BEGIN
   MachineConfig[0].Machine."Family" := 2;
   MachineConfig[0].Machine.TypeNo := 20;
   MachineConfig[0].Machine.Range := 2;
   MachineConfig[0].Machine.SepType := 1;
   MachineConfig[0].Machine.Frame := 4;
   MachineConfig[0].Machine.DchSystem := 1;
   MachineConfig[0].Machine.Spare_1 := 3;
   MachineConfig[0].Machine.FeedPump := 1;
   MachineConfig[0].Machine.eWON := 1;
   MachineConfig[0]."Unit Sep"."EM - 100"."L-GREEN".CW.ENABLE := TRUE;
   MachineConfig[0]."Unit Sep"."EM - 100"."L-YELLOW".Tag := 'L-BLUE';
   MachineConfig[0]."Unit Sep"."EM - 100".EMS.Address := 180;
   MachineConfig[0]."Unit Sep"."EM - 100".UPS.CW.ENABLE := False;
   MachineConfig[0]."Unit Sep"."EM - 100".EWON.CW.ENABLE := True;
   MachineConfig[0]."Unit Sep"."EM - 100".EWON.CW.EXIST := True;
   MachineConfig[0]."Unit Sep"."EM - 100"."LT BUF".CW.ENABLE := False;
   MachineConfig[0]."Unit Sep"."EM - 400"."AV409-1".CW.ENABLE := False;
   MachineConfig[0]."Unit Sep"."EM - 400"."AV409-1".ACT_OUT_ADD := 8;
   MachineConfig[0]."Unit Sep"."EM - 400"."FCV409-1".CW.ENABLE := False;
   MachineConfig[0]."Unit Sep"."EM - 400"."FIS409-1".CW.ENABLE := false;
   MachineConfig[0]."Unit Sep"."EM - 400"."FIT409-1".CW.ENABLE := False;
   MachineConfig[0]."Unit Sep"."EM - 701".M701."TYPE" := 2;
   MachineConfig[0]."Unit Sep"."EM - 701".M701.FB_RUN_ADD := 8;
   MachineConfig[0]."Unit Sep"."EM - 701".M701.FB_RDY_ADD := 8;
   MachineConfig[0]."Unit Sep"."EM - 701".M701.OUT_ACT_ADD := 512;
   MachineConfig[0]."Unit Sep"."EM - 701".M701.OUT_RST_ADD := 8;
   MachineConfig[0]."Unit Sep"."EM - 730".TS730.CW.ENABLE := True;
   MachineConfig[0]."Unit Sep"."EM - 730".TS730.Address := 184;
   MachineConfig[0]."Unit Sep"."EM - 740"."P+F PS".Address := 180;
   MachineConfig[0]."Unit Sep"."EM - 740"."P+F OS".Address := 182;
   MachineConfig[0]."Unit Sep"."EM - 740"."P+F ERROR".Address := 183;
   MachineConfig[0]."Unit Sep"."EM - 750".YT75X.CW.ENABLE := False;
   MachineConfig[0]."Unit Process"."EM - 201"."AV201-1".CW.ENABLE := True;
   MachineConfig[0]."Unit Process"."EM - 201"."AV201-1".CW.FB_CLS_EN := False;
   MachineConfig[0]."Unit Process"."EM - 201"."AV201-1".CW.FB_OPN_EN := False;
   MachineConfig[0]."Unit Process"."EM - 201"."AV201-1".CW.VLV_W_FB := False;
   MachineConfig[0]."Unit Process"."EM - 201"."AV201-1".FB_OPN_ADD := 8;
   MachineConfig[0]."Unit Process"."EM - 201"."AV201-1".FB_CLS_ADD := 8;
   MachineConfig[0]."Unit Process"."EM - 201"."AV201-1".ACT_OUT_ADD := 160;
   MachineConfig[0]."Unit Process"."EM - 201"."FCV201-1".CW.ENABLE := false;
   MachineConfig[0]."Unit Process"."EM - 201"."FIT201-1"."Type" := 0;
   MachineConfig[0]."Unit Process"."EM - 201"."FIT201-1".Address := 88;
   MachineConfig[0]."Unit Process"."EM - 201"."FIT201-1".Max := 10000.0;
   MachineConfig[0]."Unit Process"."EM - 201"."LA201-1".CW.ENABLE := False;
   MachineConfig[0]."Unit Process"."EM - 201"."PIT201-1".CW.ENABLE := False;
   MachineConfig[0]."Unit Process"."EM - 22X"."AV220-1".CW.ENABLE := True;
   MachineConfig[0]."Unit Process"."EM - 22X"."AV220-1".CW.FB_CLS_EN := false;
   MachineConfig[0]."Unit Process"."EM - 22X"."AV220-1".CW.FB_OPN_EN := false;
   MachineConfig[0]."Unit Process"."EM - 22X"."AV220-1".CW.EXIST := False;
   MachineConfig[0]."Unit Process"."EM - 22X"."AV220-1".CW.VLV_W_FB := false;
   MachineConfig[0]."Unit Process"."EM - 22X"."AV220-1".FB_OPN_ADD := 8;
   MachineConfig[0]."Unit Process"."EM - 22X"."AV220-1".FB_CLS_ADD := 8;
   MachineConfig[0]."Unit Process"."EM - 22X"."AV220-1".ACT_OUT_ADD := 162;
   MachineConfig[0]."Unit Process"."EM - 22X"."AV460-1".CW.ENABLE := True;
   MachineConfig[0]."Unit Process"."EM - 22X"."AV460-1".CW.FB_CLS_EN := false;
   MachineConfig[0]."Unit Process"."EM - 22X"."AV460-1".CW.FB_OPN_EN := false;
   MachineConfig[0]."Unit Process"."EM - 22X"."AV460-1".CW.EXIST := False;
   MachineConfig[0]."Unit Process"."EM - 22X"."AV460-1".CW.VLV_W_FB := false;
   MachineConfig[0]."Unit Process"."EM - 22X"."AV460-1".FB_OPN_ADD := 8;
   MachineConfig[0]."Unit Process"."EM - 22X"."AV460-1".FB_CLS_ADD := 8;
   MachineConfig[0]."Unit Process"."EM - 22X"."AV460-1".ACT_OUT_ADD := 171;
   MachineConfig[0]."Unit Process"."EM - 22X"."FIT22X-1".CW.ENABLE := False;
   MachineConfig[0]."Unit Process"."EM - 22X"."PIT22X-1".CW.ENABLE := False;
   MachineConfig[0]."Unit Process"."EM - 22X"."PIT22X-1".CW.EXIST := False;
   MachineConfig[0]."Unit Process"."EM - 22X"."QT220-1".Tag := 'QT220-1';
   MachineConfig[0]."Unit Process"."EM - 22X"."QT220-1".CW.ENABLE := True;
   MachineConfig[0]."Unit Process"."EM - 22X"."QT220-1".CW.EXIST := False;
   MachineConfig[0]."Unit Process"."EM - 22X"."QT220-1".Address := 70;
   MachineConfig[0]."Unit Process"."EM - 22X"."PCV22X-1".CW.ENABLE := False;
   MachineConfig[0]."Unit Process"."EM - 22Y"."AV221-1".CW.ENABLE := false;
   MachineConfig[0]."Unit Process"."EM - 22Y"."AV461-1".CW.ENABLE := false;
   MachineConfig[0]."Unit Process"."EM - 22Y"."FIT22Y-1".CW.ENABLE := false;
   MachineConfig[0]."Unit Process"."EM - 22Y"."LA221-1".CW.ENABLE := false;
   MachineConfig[0]."Unit Process"."EM - 22Y"."PCV22Y-1".CW.ENABLE := false;
   MachineConfig[0]."Unit Process"."EM - 22Y"."PIT22Y-1".CW.ENABLE := false;
   MachineConfig[0]."Unit Process"."EM - 340"."AV340-1".CW.ENABLE := True;
   MachineConfig[0]."Unit Process"."EM - 340"."AV340-1".CW.FB_CLS_EN := False;
   MachineConfig[0]."Unit Process"."EM - 340"."AV340-1".CW.FB_OPN_EN := False;
   MachineConfig[0]."Unit Process"."EM - 340"."AV340-1".CW.EXIST := False;
   MachineConfig[0]."Unit Process"."EM - 340"."AV340-1".CW.VLV_W_FB := False;
   MachineConfig[0]."Unit Process"."EM - 340"."AV340-1".FB_OPN_ADD := 8;
   MachineConfig[0]."Unit Process"."EM - 340"."AV340-1".FB_CLS_ADD := 8;
   MachineConfig[0]."Unit Process"."EM - 340"."AV340-1".ACT_OUT_ADD := 165;
   MachineConfig[0]."Unit Process"."EM - 340"."PIS340-1".Tag := 'PS301-1';
   MachineConfig[0]."Unit Process"."EM - 340"."PIS340-1".CW.ENABLE := True;
   MachineConfig[0]."Unit Process"."EM - 340"."V340-1".CW.ENABLE := True;
   MachineConfig[0]."Unit Process"."EM - 340"."V340-1".Address := 170;
   MachineConfig[0]."Unit Dch"."EM - 222"."LS222-1".CW.ENABLE := False;
   MachineConfig[0]."Unit Dch"."EM - 222"."P222-1".CW.EXIST := False;
   MachineConfig[0]."Unit Dch"."EM - 222"."P222-1".FB_RUN_ADD := 194;
   MachineConfig[0]."Unit Dch"."EM - 222"."P222-1".FB_RDY_ADD := 195;
   MachineConfig[0]."Unit Dch"."EM - 222"."P222-1".OUT_ACT_ADD := 182;
   MachineConfig[0]."Unit Dch"."EM - 222"."TS222-1".CW.ENABLE := false;
   MachineConfig[0]."Unit Dch"."EM - 300"."AV301-1".CW.ENABLE := True;
   MachineConfig[0]."Unit Dch"."EM - 300"."AV301-1".CW.FB_CLS_EN := false;
   MachineConfig[0]."Unit Dch"."EM - 300"."AV301-1".CW.FB_OPN_EN := false;
   MachineConfig[0]."Unit Dch"."EM - 300"."AV301-1".CW.VLV_W_FB := false;
   MachineConfig[0]."Unit Dch"."EM - 300"."AV301-1".FB_OPN_ADD := 8;
   MachineConfig[0]."Unit Dch"."EM - 300"."AV301-1".FB_CLS_ADD := 8;
   MachineConfig[0]."Unit Dch"."EM - 300"."AV301-1".ACT_OUT_ADD := 163;
   MachineConfig[0]."Unit Dch"."EM - 300"."AV304-1".TAG := 'AV301-1';
   MachineConfig[0]."Unit Dch"."EM - 300"."AV304-1".ACT_OUT_ADD := 163;
   MachineConfig[0]."Unit Dch"."EM - 300"."AV320-1".CW.ENABLE := True;
   MachineConfig[0]."Unit Dch"."EM - 300"."AV320-1".CW.FB_CLS_EN := false;
   MachineConfig[0]."Unit Dch"."EM - 300"."AV320-1".CW.FB_OPN_EN := false;
   MachineConfig[0]."Unit Dch"."EM - 300"."AV320-1".CW.EXIST := false;
   MachineConfig[0]."Unit Dch"."EM - 300"."AV320-1".CW.VLV_W_FB := false;
   MachineConfig[0]."Unit Dch"."EM - 300"."AV320-1".FB_OPN_ADD := 8;
   MachineConfig[0]."Unit Dch"."EM - 300"."AV320-1".FB_CLS_ADD := 8;
   MachineConfig[0]."Unit Dch"."EM - 300"."AV320-1".ACT_OUT_ADD := 164;
   MachineConfig[0]."Unit Dch"."EM - 300"."PS301-1".CW.ENABLE := True;
   MachineConfig[0]."Unit Dch"."EM - 375"."AV37X-1".TAG := 'AV376-1';
   MachineConfig[0]."Unit Dch"."EM - 375"."AV37X-1".CW.ENABLE := true;
   MachineConfig[0]."Unit Dch"."EM - 375"."AV37X-1".ACT_OUT_ADD := 166;
   MachineConfig[0]."Unit Dch"."EM - 375".LS793.CW.ENABLE := true;
   MachineConfig[0]."Unit Dch"."EM - 375"."PIS375-1".CW.ENABLE := false;
   MachineConfig[0]."Unit Dch"."EM - 506".IP506a.CW.ENABLE := False;
   MachineConfig[0]."Unit Dch"."EM - 506".AVDCH.TAG := 'AV372-1';
   MachineConfig[0]."Unit Dch"."EM - 506".AVDCH.CW.ENABLE := true;
   MachineConfig[0]."Unit Dch"."EM - 506".AVDCH.ACT_OUT_ADD := 167;
   MachineConfig[0].Options."EM - P201"."P201-1".FB_RUN_ADD := 196;
   MachineConfig[0].Options."EM - P201"."P201-1".FB_RDY_ADD := 197;
   MachineConfig[0].Options."EM - P201"."P201-1".OUT_ACT_ADD := 183;
   MachineConfig[0].Options."EM - P201"."P201-1".OUT_RST_ADD := 184;
   MachineConfig[0].Options."EM - P201"."P201-1_SPEED_REF".Address := 70;
   MachineConfig[1].Machine."Family" := 2;
   MachineConfig[1].Machine.TypeNo := 21;
   MachineConfig[1].Machine.Range := 2;
   MachineConfig[1].Machine.SepType := 2;
   MachineConfig[1].Machine.Frame := 4;
   MachineConfig[1].Machine.DchSystem := 1;
   MachineConfig[1].Machine.Spare_1 := 3;
   MachineConfig[1].Machine.FeedPump := 1;
   MachineConfig[1].Machine.eWON := 1;
   MachineConfig[1]."Unit Sep"."EM - 100"."L-GREEN".CW.ENABLE := True;
   MachineConfig[1]."Unit Sep"."EM - 100"."L-YELLOW".Tag := 'L-BLUE';
   MachineConfig[1]."Unit Sep"."EM - 100".EMS.Address := 180;
   MachineConfig[1]."Unit Sep"."EM - 100".UPS.CW.ENABLE := False;
   MachineConfig[1]."Unit Sep"."EM - 100".EWON.CW.ENABLE := True;
   MachineConfig[1]."Unit Sep"."EM - 100".EWON.CW.EXIST := True;
   MachineConfig[1]."Unit Sep"."EM - 100"."LT BUF".CW.ENABLE := False;
   MachineConfig[1]."Unit Sep"."EM - 400"."AV409-1".CW.ENABLE := False;
   MachineConfig[1]."Unit Sep"."EM - 400"."FCV409-1".CW.ENABLE := False;
   MachineConfig[1]."Unit Sep"."EM - 400"."FIS409-1".CW.ENABLE := false;
   MachineConfig[1]."Unit Sep"."EM - 400"."FIT409-1".CW.ENABLE := False;
   MachineConfig[1]."Unit Sep"."EM - 701".M701."TYPE" := 2;
   MachineConfig[1]."Unit Sep"."EM - 701".M701.FB_RUN_ADD := 8;
   MachineConfig[1]."Unit Sep"."EM - 701".M701.FB_RDY_ADD := 8;
   MachineConfig[1]."Unit Sep"."EM - 701".M701.OUT_ACT_ADD := 512;
   MachineConfig[1]."Unit Sep"."EM - 701".M701.OUT_RST_ADD := 8;
   MachineConfig[1]."Unit Sep"."EM - 730".TS730.CW.ENABLE := True;
   MachineConfig[1]."Unit Sep"."EM - 730".TS730.Address := 184;
   MachineConfig[1]."Unit Sep"."EM - 740"."P+F PS".Address := 180;
   MachineConfig[1]."Unit Sep"."EM - 740"."P+F OS".Address := 182;
   MachineConfig[1]."Unit Sep"."EM - 740"."P+F ERROR".Address := 183;
   MachineConfig[1]."Unit Sep"."EM - 750".YT75X.CW.ENABLE := False;
   MachineConfig[1]."Unit Process"."EM - 201"."AV201-1".CW.ENABLE := True;
   MachineConfig[1]."Unit Process"."EM - 201"."AV201-1".CW.VLV_W_FB := false;
   MachineConfig[1]."Unit Process"."EM - 201"."AV201-1".FB_OPN_ADD := 8;
   MachineConfig[1]."Unit Process"."EM - 201"."AV201-1".FB_CLS_ADD := 8;
   MachineConfig[1]."Unit Process"."EM - 201"."AV201-1".ACT_OUT_ADD := 160;
   MachineConfig[1]."Unit Process"."EM - 201"."FCV201-1".CW.ENABLE := false;
   MachineConfig[1]."Unit Process"."EM - 201"."FIT201-1"."Type" := 0;
   MachineConfig[1]."Unit Process"."EM - 201"."FIT201-1".Address := 88;
   MachineConfig[1]."Unit Process"."EM - 201"."FIT201-1".Max := 10000.0;
   MachineConfig[1]."Unit Process"."EM - 201"."LA201-1".CW.ENABLE := False;
   MachineConfig[1]."Unit Process"."EM - 201"."PIT201-1".CW.ENABLE := False;
   MachineConfig[1]."Unit Process"."EM - 22X"."FIT22X-1".CW.ENABLE := False;
   MachineConfig[1]."Unit Process"."EM - 22X"."PIT22X-1".CW.ENABLE := False;
   MachineConfig[1]."Unit Process"."EM - 22X"."PCV22X-1".CW.ENABLE := False;
   MachineConfig[1]."Unit Process"."EM - 22Y"."AV221-1".CW.ENABLE := True;
   MachineConfig[1]."Unit Process"."EM - 22Y"."AV221-1".CW.FB_CLS_EN := false;
   MachineConfig[1]."Unit Process"."EM - 22Y"."AV221-1".CW.FB_OPN_EN := false;
   MachineConfig[1]."Unit Process"."EM - 22Y"."AV221-1".CW.EXIST := false;
   MachineConfig[1]."Unit Process"."EM - 22Y"."AV221-1".CW.VLV_W_FB := false;
   MachineConfig[1]."Unit Process"."EM - 22Y"."AV221-1".FB_OPN_ADD := 8;
   MachineConfig[1]."Unit Process"."EM - 22Y"."AV221-1".FB_CLS_ADD := 8;
   MachineConfig[1]."Unit Process"."EM - 22Y"."AV221-1".ACT_OUT_ADD := 175;
   MachineConfig[1]."Unit Process"."EM - 22Y"."AV461-1".CW.ENABLE := True;
   MachineConfig[1]."Unit Process"."EM - 22Y"."AV461-1".CW.FB_CLS_EN := false;
   MachineConfig[1]."Unit Process"."EM - 22Y"."AV461-1".CW.FB_OPN_EN := false;
   MachineConfig[1]."Unit Process"."EM - 22Y"."AV461-1".CW.EXIST := false;
   MachineConfig[1]."Unit Process"."EM - 22Y"."AV461-1".CW.VLV_W_FB := false;
   MachineConfig[1]."Unit Process"."EM - 22Y"."AV461-1".FB_OPN_ADD := 8;
   MachineConfig[1]."Unit Process"."EM - 22Y"."AV461-1".FB_CLS_ADD := 8;
   MachineConfig[1]."Unit Process"."EM - 22Y"."AV461-1".ACT_OUT_ADD := 176;
   MachineConfig[1]."Unit Process"."EM - 340"."AV340-1".CW.FB_CLS_EN := False;
   MachineConfig[1]."Unit Process"."EM - 340"."AV340-1".CW.FB_OPN_EN := False;
   MachineConfig[1]."Unit Process"."EM - 340"."AV340-1".CW.EXIST := False;
   MachineConfig[1]."Unit Process"."EM - 340"."AV340-1".CW.VLV_W_FB := False;
   MachineConfig[1]."Unit Process"."EM - 340"."AV340-1".FB_OPN_ADD := 8;
   MachineConfig[1]."Unit Process"."EM - 340"."AV340-1".FB_CLS_ADD := 8;
   MachineConfig[1]."Unit Process"."EM - 340"."AV340-1".ACT_OUT_ADD := 165;
   MachineConfig[1]."Unit Process"."EM - 340"."PIS340-1".Tag := 'PS301-1';
   MachineConfig[1]."Unit Process"."EM - 340"."PIS340-1".CW.ENABLE := True;
   MachineConfig[1]."Unit Dch"."EM - 222"."LS222-1".CW.ENABLE := False;
   MachineConfig[1]."Unit Dch"."EM - 222"."P222-1".CW.EXIST := False;
   MachineConfig[1]."Unit Dch"."EM - 222"."P222-1".FB_RUN_ADD := 194;
   MachineConfig[1]."Unit Dch"."EM - 222"."P222-1".FB_RDY_ADD := 195;
   MachineConfig[1]."Unit Dch"."EM - 222"."P222-1".OUT_ACT_ADD := 182;
   MachineConfig[1]."Unit Dch"."EM - 222"."TS222-1".CW.ENABLE := False;
   MachineConfig[1]."Unit Dch"."EM - 300"."AV301-1".CW.ENABLE := True;
   MachineConfig[1]."Unit Dch"."EM - 300"."AV301-1".CW.FB_CLS_EN := false;
   MachineConfig[1]."Unit Dch"."EM - 300"."AV301-1".CW.FB_OPN_EN := false;
   MachineConfig[1]."Unit Dch"."EM - 300"."AV301-1".CW.VLV_W_FB := false;
   MachineConfig[1]."Unit Dch"."EM - 300"."AV301-1".FB_OPN_ADD := 8;
   MachineConfig[1]."Unit Dch"."EM - 300"."AV301-1".FB_CLS_ADD := 8;
   MachineConfig[1]."Unit Dch"."EM - 300"."AV301-1".ACT_OUT_ADD := 163;
   MachineConfig[1]."Unit Dch"."EM - 300"."AV304-1".TAG := 'AV301-1';
   MachineConfig[1]."Unit Dch"."EM - 300"."AV304-1".ACT_OUT_ADD := 163;
   MachineConfig[1]."Unit Dch"."EM - 300"."AV320-1".CW.ENABLE := True;
   MachineConfig[1]."Unit Dch"."EM - 300"."AV320-1".CW.FB_CLS_EN := False;
   MachineConfig[1]."Unit Dch"."EM - 300"."AV320-1".CW.FB_OPN_EN := False;
   MachineConfig[1]."Unit Dch"."EM - 300"."AV320-1".CW.EXIST := False;
   MachineConfig[1]."Unit Dch"."EM - 300"."AV320-1".CW.VLV_W_FB := False;
   MachineConfig[1]."Unit Dch"."EM - 300"."AV320-1".FB_OPN_ADD := 8;
   MachineConfig[1]."Unit Dch"."EM - 300"."AV320-1".FB_CLS_ADD := 8;
   MachineConfig[1]."Unit Dch"."EM - 300"."AV320-1".ACT_OUT_ADD := 164;
   MachineConfig[1]."Unit Dch"."EM - 300"."PS301-1".CW.ENABLE := True;
   MachineConfig[1]."Unit Dch"."EM - 375"."AV37X-1".TAG := 'AV376-1';
   MachineConfig[1]."Unit Dch"."EM - 375"."AV37X-1".CW.ENABLE := true;
   MachineConfig[1]."Unit Dch"."EM - 375"."AV37X-1".ACT_OUT_ADD := 166;
   MachineConfig[1]."Unit Dch"."EM - 375".LS793.CW.ENABLE := true;
   MachineConfig[1]."Unit Dch"."EM - 375"."PIS375-1".CW.ENABLE := false;
   MachineConfig[1]."Unit Dch"."EM - 506".IP506a.CW.ENABLE := False;
   MachineConfig[1]."Unit Dch"."EM - 506".AVDCH.TAG := 'AV372-1';
   MachineConfig[1]."Unit Dch"."EM - 506".AVDCH.ACT_OUT_ADD := 167;
   MachineConfig[1].Options."EM - P201"."P201-1".FB_RUN_ADD := 196;
   MachineConfig[1].Options."EM - P201"."P201-1".FB_RDY_ADD := 197;
   MachineConfig[1].Options."EM - P201"."P201-1".OUT_ACT_ADD := 183;
   MachineConfig[1].Options."EM - P201"."P201-1".OUT_RST_ADD := 184;
   MachineConfig[1].Options."EM - P201"."P201-1_SPEED_REF".Address := 70;
   MachineConfig[2].Machine."Family" := 2;
   MachineConfig[2].Machine.TypeNo := 22;
   MachineConfig[2].Machine.Range := 2;
   MachineConfig[2].Machine.SepType := 3;
   MachineConfig[2].Machine.Frame := 4;
   MachineConfig[2].Machine.DchSystem := 1;
   MachineConfig[2].Machine.Spare_1 := 3;
   MachineConfig[2].Machine.FeedPump := 1;
   MachineConfig[2].Machine.eWON := 1;
   MachineConfig[2]."Unit Sep"."EM - 100"."L-GREEN".CW.ENABLE := True;
   MachineConfig[2]."Unit Sep"."EM - 100"."L-YELLOW".Tag := 'L-BLUE';
   MachineConfig[2]."Unit Sep"."EM - 100".EMS.Address := 180;
   MachineConfig[2]."Unit Sep"."EM - 100".UPS.CW.ENABLE := False;
   MachineConfig[2]."Unit Sep"."EM - 100".EWON.CW.ENABLE := True;
   MachineConfig[2]."Unit Sep"."EM - 100".EWON.CW.EXIST := True;
   MachineConfig[2]."Unit Sep"."EM - 100"."LT BUF".CW.ENABLE := False;
   MachineConfig[2]."Unit Sep"."EM - 400"."AV409-1".CW.ENABLE := False;
   MachineConfig[2]."Unit Sep"."EM - 400"."FCV409-1".CW.ENABLE := False;
   MachineConfig[2]."Unit Sep"."EM - 400"."FIS409-1".CW.ENABLE := false;
   MachineConfig[2]."Unit Sep"."EM - 400"."FIT409-1".CW.ENABLE := False;
   MachineConfig[2]."Unit Sep"."EM - 701".M701."TYPE" := 2;
   MachineConfig[2]."Unit Sep"."EM - 701".M701.FB_RUN_ADD := 8;
   MachineConfig[2]."Unit Sep"."EM - 701".M701.FB_RDY_ADD := 8;
   MachineConfig[2]."Unit Sep"."EM - 701".M701.OUT_ACT_ADD := 512;
   MachineConfig[2]."Unit Sep"."EM - 701".M701.OUT_RST_ADD := 8;
   MachineConfig[2]."Unit Sep"."EM - 730".TS730.CW.ENABLE := True;
   MachineConfig[2]."Unit Sep"."EM - 730".TS730.Address := 184;
   MachineConfig[2]."Unit Sep"."EM - 740"."P+F PS".Address := 180;
   MachineConfig[2]."Unit Sep"."EM - 740"."P+F OS".Address := 182;
   MachineConfig[2]."Unit Sep"."EM - 740"."P+F ERROR".Address := 183;
   MachineConfig[2]."Unit Sep"."EM - 750".YT75X.CW.ENABLE := False;
   MachineConfig[2]."Unit Process"."EM - 201"."AV201-1".CW.ENABLE := True;
   MachineConfig[2]."Unit Process"."EM - 201"."AV201-1".CW.FB_CLS_EN := False;
   MachineConfig[2]."Unit Process"."EM - 201"."AV201-1".CW.FB_OPN_EN := False;
   MachineConfig[2]."Unit Process"."EM - 201"."AV201-1".CW.VLV_W_FB := False;
   MachineConfig[2]."Unit Process"."EM - 201"."AV201-1".FB_OPN_ADD := 8;
   MachineConfig[2]."Unit Process"."EM - 201"."AV201-1".FB_CLS_ADD := 8;
   MachineConfig[2]."Unit Process"."EM - 201"."AV201-1".ACT_OUT_ADD := 160;
   MachineConfig[2]."Unit Process"."EM - 201"."FCV201-1".CW.ENABLE := false;
   MachineConfig[2]."Unit Process"."EM - 201"."FIT201-1"."Type" := 0;
   MachineConfig[2]."Unit Process"."EM - 201"."FIT201-1".Address := 88;
   MachineConfig[2]."Unit Process"."EM - 201"."FIT201-1".Max := 10000.0;
   MachineConfig[2]."Unit Process"."EM - 201"."LA201-1".CW.ENABLE := False;
   MachineConfig[2]."Unit Process"."EM - 201"."PIT201-1".CW.ENABLE := False;
   MachineConfig[2]."Unit Process"."EM - 22X"."FIT22X-1".CW.ENABLE := False;
   MachineConfig[2]."Unit Process"."EM - 22X"."PIT22X-1".CW.ENABLE := False;
   MachineConfig[2]."Unit Process"."EM - 22X"."PCV22X-1".CW.ENABLE := False;
   MachineConfig[2]."Unit Process"."EM - 22Y"."AV221-1".CW.ENABLE := True;
   MachineConfig[2]."Unit Process"."EM - 22Y"."AV221-1".CW.FB_CLS_EN := False;
   MachineConfig[2]."Unit Process"."EM - 22Y"."AV221-1".CW.FB_OPN_EN := False;
   MachineConfig[2]."Unit Process"."EM - 22Y"."AV221-1".CW.EXIST := False;
   MachineConfig[2]."Unit Process"."EM - 22Y"."AV221-1".CW.VLV_W_FB := False;
   MachineConfig[2]."Unit Process"."EM - 22Y"."AV221-1".FB_OPN_ADD := 8;
   MachineConfig[2]."Unit Process"."EM - 22Y"."AV221-1".FB_CLS_ADD := 8;
   MachineConfig[2]."Unit Process"."EM - 22Y"."AV221-1".ACT_OUT_ADD := 175;
   MachineConfig[2]."Unit Process"."EM - 22Y"."AV461-1".CW.ENABLE := True;
   MachineConfig[2]."Unit Process"."EM - 22Y"."AV461-1".CW.FB_CLS_EN := False;
   MachineConfig[2]."Unit Process"."EM - 22Y"."AV461-1".CW.FB_OPN_EN := False;
   MachineConfig[2]."Unit Process"."EM - 22Y"."AV461-1".CW.EXIST := False;
   MachineConfig[2]."Unit Process"."EM - 22Y"."AV461-1".CW.VLV_W_FB := False;
   MachineConfig[2]."Unit Process"."EM - 22Y"."AV461-1".FB_OPN_ADD := 8;
   MachineConfig[2]."Unit Process"."EM - 22Y"."AV461-1".FB_CLS_ADD := 8;
   MachineConfig[2]."Unit Process"."EM - 22Y"."AV461-1".ACT_OUT_ADD := 176;
   MachineConfig[2]."Unit Process"."EM - 22Y"."QT221-1".Tag := 'QT221-1';
   MachineConfig[2]."Unit Process"."EM - 22Y"."QT221-1".CW.ENABLE := True;
   MachineConfig[2]."Unit Process"."EM - 22Y"."QT221-1".Address := 70;
   MachineConfig[2]."Unit Process"."EM - 340"."AV340-1".CW.FB_CLS_EN := False;
   MachineConfig[2]."Unit Process"."EM - 340"."AV340-1".CW.FB_OPN_EN := False;
   MachineConfig[2]."Unit Process"."EM - 340"."AV340-1".CW.EXIST := False;
   MachineConfig[2]."Unit Process"."EM - 340"."AV340-1".CW.VLV_W_FB := False;
   MachineConfig[2]."Unit Process"."EM - 340"."AV340-1".FB_OPN_ADD := 8;
   MachineConfig[2]."Unit Process"."EM - 340"."AV340-1".FB_CLS_ADD := 8;
   MachineConfig[2]."Unit Process"."EM - 340"."AV340-1".ACT_OUT_ADD := 165;
   MachineConfig[2]."Unit Process"."EM - 340"."PIS340-1".Tag := 'PS301-1';
   MachineConfig[2]."Unit Process"."EM - 340"."PIS340-1".CW.ENABLE := True;
   MachineConfig[2]."Unit Dch"."EM - 222"."LS222-1".CW.ENABLE := False;
   MachineConfig[2]."Unit Dch"."EM - 222"."P222-1".CW.EXIST := False;
   MachineConfig[2]."Unit Dch"."EM - 222"."P222-1".FB_RUN_ADD := 194;
   MachineConfig[2]."Unit Dch"."EM - 222"."P222-1".FB_RDY_ADD := 195;
   MachineConfig[2]."Unit Dch"."EM - 222"."P222-1".OUT_ACT_ADD := 182;
   MachineConfig[2]."Unit Dch"."EM - 222"."TS222-1".CW.ENABLE := False;
   MachineConfig[2]."Unit Dch"."EM - 300"."AV301-1".CW.ENABLE := True;
   MachineConfig[2]."Unit Dch"."EM - 300"."AV301-1".CW.FB_CLS_EN := false;
   MachineConfig[2]."Unit Dch"."EM - 300"."AV301-1".CW.FB_OPN_EN := false;
   MachineConfig[2]."Unit Dch"."EM - 300"."AV301-1".CW.VLV_W_FB := false;
   MachineConfig[2]."Unit Dch"."EM - 300"."AV301-1".FB_OPN_ADD := 8;
   MachineConfig[2]."Unit Dch"."EM - 300"."AV301-1".FB_CLS_ADD := 8;
   MachineConfig[2]."Unit Dch"."EM - 300"."AV301-1".ACT_OUT_ADD := 163;
   MachineConfig[2]."Unit Dch"."EM - 300"."AV304-1".TAG := 'AV301-1';
   MachineConfig[2]."Unit Dch"."EM - 300"."AV304-1".ACT_OUT_ADD := 163;
   MachineConfig[2]."Unit Dch"."EM - 300"."AV320-1".CW.ENABLE := True;
   MachineConfig[2]."Unit Dch"."EM - 300"."AV320-1".CW.FB_CLS_EN := False;
   MachineConfig[2]."Unit Dch"."EM - 300"."AV320-1".CW.FB_OPN_EN := False;
   MachineConfig[2]."Unit Dch"."EM - 300"."AV320-1".CW.EXIST := False;
   MachineConfig[2]."Unit Dch"."EM - 300"."AV320-1".CW.VLV_W_FB := False;
   MachineConfig[2]."Unit Dch"."EM - 300"."AV320-1".FB_OPN_ADD := 8;
   MachineConfig[2]."Unit Dch"."EM - 300"."AV320-1".FB_CLS_ADD := 8;
   MachineConfig[2]."Unit Dch"."EM - 300"."AV320-1".ACT_OUT_ADD := 164;
   MachineConfig[2]."Unit Dch"."EM - 300"."PS301-1".CW.ENABLE := True;
   MachineConfig[2]."Unit Dch"."EM - 375"."AV37X-1".TAG := 'AV376-1';
   MachineConfig[2]."Unit Dch"."EM - 375"."AV37X-1".CW.ENABLE := true;
   MachineConfig[2]."Unit Dch"."EM - 375"."AV37X-1".ACT_OUT_ADD := 166;
   MachineConfig[2]."Unit Dch"."EM - 375".LS793.CW.ENABLE := true;
   MachineConfig[2]."Unit Dch"."EM - 375"."PIS375-1".CW.ENABLE := false;
   MachineConfig[2]."Unit Dch"."EM - 506".IP506a.CW.ENABLE := False;
   MachineConfig[2]."Unit Dch"."EM - 506".AVDCH.TAG := 'AV372-1';
   MachineConfig[2]."Unit Dch"."EM - 506".AVDCH.CW.ENABLE := true;
   MachineConfig[2]."Unit Dch"."EM - 506".AVDCH.ACT_OUT_ADD := 167;
   MachineConfig[2].Options."EM - P201"."P201-1".FB_RUN_ADD := 196;
   MachineConfig[2].Options."EM - P201"."P201-1".FB_RDY_ADD := 197;
   MachineConfig[2].Options."EM - P201"."P201-1".OUT_ACT_ADD := 183;
   MachineConfig[2].Options."EM - P201"."P201-1".OUT_RST_ADD := 184;
   MachineConfig[2].Options."EM - P201"."P201-1_SPEED_REF".Address := 70;
   MachineConfig[3].Machine."Family" := 2;
   MachineConfig[3].Machine.TypeNo := 23;
   MachineConfig[3].Machine.Range := 2;
   MachineConfig[3].Machine.SepType := 1;
   MachineConfig[3].Machine.Frame := 6;
   MachineConfig[3].Machine.DchSystem := 1;
   MachineConfig[3].Machine.FeedPump := 1;
   MachineConfig[3].Machine.eWON := 1;
   MachineConfig[3]."Unit Sep"."EM - 100"."L-GREEN".CW.ENABLE := True;
   MachineConfig[3]."Unit Sep"."EM - 100"."L-YELLOW".Tag := 'L-BLUE';
   MachineConfig[3]."Unit Sep"."EM - 100".EMS.Address := 180;
   MachineConfig[3]."Unit Sep"."EM - 100".UPS.CW.ENABLE := False;
   MachineConfig[3]."Unit Sep"."EM - 100".EWON.CW.ENABLE := True;
   MachineConfig[3]."Unit Sep"."EM - 100".EWON.CW.EXIST := True;
   MachineConfig[3]."Unit Sep"."EM - 400"."AV409-1".CW.ENABLE := False;
   MachineConfig[3]."Unit Sep"."EM - 400"."FCV409-1".CW.ENABLE := False;
   MachineConfig[3]."Unit Sep"."EM - 400"."FIS409-1".CW.ENABLE := false;
   MachineConfig[3]."Unit Sep"."EM - 400"."FIT409-1".CW.ENABLE := False;
   MachineConfig[3]."Unit Sep"."EM - 600"."FIS615-1".CW.ENABLE := False;
   MachineConfig[3]."Unit Sep"."EM - 701".M701."TYPE" := 2;
   MachineConfig[3]."Unit Sep"."EM - 701".M701.FB_RUN_ADD := 8;
   MachineConfig[3]."Unit Sep"."EM - 701".M701.FB_RDY_ADD := 8;
   MachineConfig[3]."Unit Sep"."EM - 701".M701.OUT_ACT_ADD := 512;
   MachineConfig[3]."Unit Sep"."EM - 701".M701.OUT_RST_ADD := 8;
   MachineConfig[3]."Unit Sep"."EM - 730".TS730.CW.ENABLE := True;
   MachineConfig[3]."Unit Sep"."EM - 730".TS730.Address := 184;
   MachineConfig[3]."Unit Sep"."EM - 740"."P+F PS".Address := 180;
   MachineConfig[3]."Unit Sep"."EM - 740"."P+F OS".Address := 182;
   MachineConfig[3]."Unit Sep"."EM - 740"."P+F ERROR".Address := 183;
   MachineConfig[3]."Unit Sep"."EM - 750".YT75X.Tag := 'YT752';
   MachineConfig[3]."Unit Sep"."EM - 750".YT75X.CW.ENABLE := True;
   MachineConfig[3]."Unit Sep"."EM - 750".YT75X.Address := 78;
   MachineConfig[3]."Unit Sep"."EM - 750".YT75X.Min := 2.3;
   MachineConfig[3]."Unit Sep"."EM - 750".YT75X.Max := 5.5;
   MachineConfig[3]."Unit Process"."EM - 201"."AV201-1".CW.ENABLE := True;
   MachineConfig[3]."Unit Process"."EM - 201"."AV201-1".CW.FB_CLS_EN := False;
   MachineConfig[3]."Unit Process"."EM - 201"."AV201-1".CW.FB_OPN_EN := False;
   MachineConfig[3]."Unit Process"."EM - 201"."AV201-1".CW.VLV_W_FB := False;
   MachineConfig[3]."Unit Process"."EM - 201"."AV201-1".FB_OPN_ADD := 8;
   MachineConfig[3]."Unit Process"."EM - 201"."AV201-1".FB_CLS_ADD := 8;
   MachineConfig[3]."Unit Process"."EM - 201"."AV201-1".ACT_OUT_ADD := 160;
   MachineConfig[3]."Unit Process"."EM - 201"."FCV201-1".CW.ENABLE := false;
   MachineConfig[3]."Unit Process"."EM - 201"."FIT201-1"."Type" := 0;
   MachineConfig[3]."Unit Process"."EM - 201"."FIT201-1".Address := 88;
   MachineConfig[3]."Unit Process"."EM - 201"."FIT201-1".Max := 10000.0;
   MachineConfig[3]."Unit Process"."EM - 201"."LA201-1".CW.ENABLE := False;
   MachineConfig[3]."Unit Process"."EM - 201"."PIT201-1".CW.ENABLE := true;
   MachineConfig[3]."Unit Process"."EM - 201"."PIT201-1".CW.EXIST := false;
   MachineConfig[3]."Unit Process"."EM - 22X"."AV220-1".CW.ENABLE := True;
   MachineConfig[3]."Unit Process"."EM - 22X"."AV220-1".CW.FB_CLS_EN := false;
   MachineConfig[3]."Unit Process"."EM - 22X"."AV220-1".CW.FB_OPN_EN := false;
   MachineConfig[3]."Unit Process"."EM - 22X"."AV220-1".CW.EXIST := false;
   MachineConfig[3]."Unit Process"."EM - 22X"."AV220-1".CW.VLV_W_FB := false;
   MachineConfig[3]."Unit Process"."EM - 22X"."AV220-1".FB_OPN_ADD := 8;
   MachineConfig[3]."Unit Process"."EM - 22X"."AV220-1".FB_CLS_ADD := 8;
   MachineConfig[3]."Unit Process"."EM - 22X"."AV220-1".ACT_OUT_ADD := 162;
   MachineConfig[3]."Unit Process"."EM - 22X"."AV460-1".CW.ENABLE := True;
   MachineConfig[3]."Unit Process"."EM - 22X"."AV460-1".CW.FB_CLS_EN := false;
   MachineConfig[3]."Unit Process"."EM - 22X"."AV460-1".CW.FB_OPN_EN := false;
   MachineConfig[3]."Unit Process"."EM - 22X"."AV460-1".CW.EXIST := false;
   MachineConfig[3]."Unit Process"."EM - 22X"."AV460-1".CW.VLV_W_FB := false;
   MachineConfig[3]."Unit Process"."EM - 22X"."AV460-1".FB_OPN_ADD := 8;
   MachineConfig[3]."Unit Process"."EM - 22X"."AV460-1".FB_CLS_ADD := 8;
   MachineConfig[3]."Unit Process"."EM - 22X"."AV460-1".ACT_OUT_ADD := 171;
   MachineConfig[3]."Unit Process"."EM - 22X"."FIT22X-1".CW.ENABLE := False;
   MachineConfig[3]."Unit Process"."EM - 22X"."PIT22X-1".CW.ENABLE := True;
   MachineConfig[3]."Unit Process"."EM - 22X"."PIT22X-1".CW.EXIST := False;
   MachineConfig[3]."Unit Process"."EM - 22X"."QT220-1".CW.ENABLE := True;
   MachineConfig[3]."Unit Process"."EM - 22X"."QT220-1".CW.EXIST := False;
   MachineConfig[3]."Unit Process"."EM - 22X"."PCV22X-1".CW.ENABLE := False;
   MachineConfig[3]."Unit Process"."EM - 340"."AV340-1".CW.ENABLE := True;
   MachineConfig[3]."Unit Process"."EM - 340"."AV340-1".CW.FB_CLS_EN := False;
   MachineConfig[3]."Unit Process"."EM - 340"."AV340-1".CW.FB_OPN_EN := False;
   MachineConfig[3]."Unit Process"."EM - 340"."AV340-1".CW.EXIST := false;
   MachineConfig[3]."Unit Process"."EM - 340"."AV340-1".CW.VLV_W_FB := False;
   MachineConfig[3]."Unit Process"."EM - 340"."AV340-1".FB_OPN_ADD := 8;
   MachineConfig[3]."Unit Process"."EM - 340"."AV340-1".FB_CLS_ADD := 8;
   MachineConfig[3]."Unit Process"."EM - 340"."AV340-1".ACT_OUT_ADD := 165;
   MachineConfig[3]."Unit Process"."EM - 340"."PIS340-1".Tag := 'PS301-1';
   MachineConfig[3]."Unit Process"."EM - 340"."PIS340-1".CW.ENABLE := True;
   MachineConfig[3]."Unit Process"."EM - 340"."V340-1".CW.ENABLE := true;
   MachineConfig[3]."Unit Process"."EM - 340"."V340-1".CW.EXIST := true;
   MachineConfig[3]."Unit Process"."EM - 340"."V340-1".Address := 170;
   MachineConfig[3]."Unit Dch"."EM - 222"."LS222-1".CW.ENABLE := False;
   MachineConfig[3]."Unit Dch"."EM - 222"."P222-1".CW.EXIST := False;
   MachineConfig[3]."Unit Dch"."EM - 222"."P222-1".FB_RUN_ADD := 194;
   MachineConfig[3]."Unit Dch"."EM - 222"."P222-1".FB_RDY_ADD := 195;
   MachineConfig[3]."Unit Dch"."EM - 222"."P222-1".OUT_ACT_ADD := 182;
   MachineConfig[3]."Unit Dch"."EM - 222"."TS222-1".CW.ENABLE := False;
   MachineConfig[3]."Unit Dch"."EM - 300"."AV301-1".CW.ENABLE := True;
   MachineConfig[3]."Unit Dch"."EM - 300"."AV301-1".CW.FB_CLS_EN := false;
   MachineConfig[3]."Unit Dch"."EM - 300"."AV301-1".CW.FB_OPN_EN := false;
   MachineConfig[3]."Unit Dch"."EM - 300"."AV301-1".CW.VLV_W_FB := false;
   MachineConfig[3]."Unit Dch"."EM - 300"."AV301-1".FB_OPN_ADD := 8;
   MachineConfig[3]."Unit Dch"."EM - 300"."AV301-1".FB_CLS_ADD := 8;
   MachineConfig[3]."Unit Dch"."EM - 300"."AV301-1".ACT_OUT_ADD := 163;
   MachineConfig[3]."Unit Dch"."EM - 300"."AV304-1".TAG := 'AV302-1';
   MachineConfig[3]."Unit Dch"."EM - 300"."AV304-1".ACT_OUT_ADD := 163;
   MachineConfig[3]."Unit Dch"."EM - 300"."AV320-1".CW.ENABLE := True;
   MachineConfig[3]."Unit Dch"."EM - 300"."AV320-1".CW.FB_CLS_EN := False;
   MachineConfig[3]."Unit Dch"."EM - 300"."AV320-1".CW.FB_OPN_EN := False;
   MachineConfig[3]."Unit Dch"."EM - 300"."AV320-1".CW.VLV_W_FB := False;
   MachineConfig[3]."Unit Dch"."EM - 300"."AV320-1".FB_OPN_ADD := 8;
   MachineConfig[3]."Unit Dch"."EM - 300"."AV320-1".FB_CLS_ADD := 8;
   MachineConfig[3]."Unit Dch"."EM - 300"."AV320-1".ACT_OUT_ADD := 164;
   MachineConfig[3]."Unit Dch"."EM - 375"."AV37X-1".TAG := 'AV376-1';
   MachineConfig[3]."Unit Dch"."EM - 375"."AV37X-1".CW.ENABLE := true;
   MachineConfig[3]."Unit Dch"."EM - 375"."AV37X-1".ACT_OUT_ADD := 166;
   MachineConfig[3]."Unit Dch"."EM - 375"."PIS375-1".CW.ENABLE := false;
   MachineConfig[3]."Unit Dch"."EM - 506".IP506a.CW.ENABLE := False;
   MachineConfig[3]."Unit Dch"."EM - 506".AVDCH.TAG := 'AV372-1';
   MachineConfig[3]."Unit Dch"."EM - 506".AVDCH.CW.ENABLE := true;
   MachineConfig[3]."Unit Dch"."EM - 506".AVDCH.ACT_OUT_ADD := 167;
   MachineConfig[3].Options."EM - P201"."P201-1".FB_RUN_ADD := 196;
   MachineConfig[3].Options."EM - P201"."P201-1".FB_RDY_ADD := 197;
   MachineConfig[3].Options."EM - P201"."P201-1".OUT_ACT_ADD := 183;
   MachineConfig[3].Options."EM - P201"."P201-1".OUT_RST_ADD := 184;
   MachineConfig[3].Options."EM - P201"."P201-1_SPEED_REF".Address := 70;
   MachineConfig[4].Machine."Family" := 2;
   MachineConfig[4].Machine.TypeNo := 24;
   MachineConfig[4].Machine.Range := 2;
   MachineConfig[4].Machine.SepType := 1;
   MachineConfig[4].Machine.Frame := 6;
   MachineConfig[4].Machine.DchSystem := 1;
   MachineConfig[4].Machine.FeedPump := 1;
   MachineConfig[4].Machine.eWON := 1;
   MachineConfig[4]."Unit Sep"."EM - 100"."L-GREEN".CW.ENABLE := True;
   MachineConfig[4]."Unit Sep"."EM - 100"."L-YELLOW".Tag := 'L-BLUE';
   MachineConfig[4]."Unit Sep"."EM - 100".EMS.Address := 180;
   MachineConfig[4]."Unit Sep"."EM - 100".UPS.CW.ENABLE := True;
   MachineConfig[4]."Unit Sep"."EM - 100".UPS.CW.EXIST := True;
   MachineConfig[4]."Unit Sep"."EM - 100".UPS.Address := 181;
   MachineConfig[4]."Unit Sep"."EM - 100".EWON.CW.ENABLE := True;
   MachineConfig[4]."Unit Sep"."EM - 100".EWON.CW.EXIST := True;
   MachineConfig[4]."Unit Sep"."EM - 400"."AV409-1".CW.ENABLE := False;
   MachineConfig[4]."Unit Sep"."EM - 400"."AV409-1".ACT_OUT_ADD := 170;
   MachineConfig[4]."Unit Sep"."EM - 400"."FIS409-1".CW.ENABLE := false;
   MachineConfig[4]."Unit Sep"."EM - 400"."TT41X-1"."Type" := 0;
   MachineConfig[4]."Unit Sep"."EM - 400"."TT41X-1".Address := 86;
   MachineConfig[4]."Unit Sep"."EM - 400"."TT41X-1".Min := -50.0;
   MachineConfig[4]."Unit Sep"."EM - 400"."TT41X-1".Max := 150.0;
   MachineConfig[4]."Unit Sep"."EM - 600"."AV63X/441-1".TAG := 'AV635-1';
   MachineConfig[4]."Unit Sep"."EM - 600"."AV63X/441-1".CW.ENABLE := True;
   MachineConfig[4]."Unit Sep"."EM - 600"."AV63X/441-1".CW.NO := True;
   MachineConfig[4]."Unit Sep"."EM - 600"."AV63X/441-1".CW.EXIST := True;
   MachineConfig[4]."Unit Sep"."EM - 600"."AV63X/441-1".ACT_OUT_ADD := 174;
   MachineConfig[4]."Unit Sep"."EM - 600"."FIS615-1".CW.ENABLE := False;
   MachineConfig[4]."Unit Sep"."EM - 600"."FIS635-1".CW.ENABLE := True;
   MachineConfig[4]."Unit Sep"."EM - 701".M701."TYPE" := 2;
   MachineConfig[4]."Unit Sep"."EM - 701".M701.FB_RUN_ADD := 8;
   MachineConfig[4]."Unit Sep"."EM - 701".M701.FB_RDY_ADD := 8;
   MachineConfig[4]."Unit Sep"."EM - 701".M701.OUT_ACT_ADD := 512;
   MachineConfig[4]."Unit Sep"."EM - 701".M701.OUT_RST_ADD := 8;
   MachineConfig[4]."Unit Sep"."EM - 730".TS730.CW.ENABLE := True;
   MachineConfig[4]."Unit Sep"."EM - 730".TS730.Address := 184;
   MachineConfig[4]."Unit Sep"."EM - 740"."P+F PS".Address := 180;
   MachineConfig[4]."Unit Sep"."EM - 740"."P+F OS".Address := 182;
   MachineConfig[4]."Unit Sep"."EM - 740"."P+F ERROR".Address := 183;
   MachineConfig[4]."Unit Sep"."EM - 750".YT75X.Tag := 'YT752';
   MachineConfig[4]."Unit Sep"."EM - 750".YT75X.CW.ENABLE := True;
   MachineConfig[4]."Unit Sep"."EM - 750".YT75X.Address := 78;
   MachineConfig[4]."Unit Sep"."EM - 750".YT75X.Min := 2.3;
   MachineConfig[4]."Unit Sep"."EM - 750".YT75X.Max := 5.5;
   MachineConfig[4]."Unit Process"."EM - 201"."AV201-1".CW.ENABLE := True;
   MachineConfig[4]."Unit Process"."EM - 201"."AV201-1".CW.FB_CLS_EN := False;
   MachineConfig[4]."Unit Process"."EM - 201"."AV201-1".CW.FB_OPN_EN := False;
   MachineConfig[4]."Unit Process"."EM - 201"."AV201-1".CW.VLV_W_FB := False;
   MachineConfig[4]."Unit Process"."EM - 201"."AV201-1".FB_OPN_ADD := 8;
   MachineConfig[4]."Unit Process"."EM - 201"."AV201-1".FB_CLS_ADD := 8;
   MachineConfig[4]."Unit Process"."EM - 201"."AV201-1".ACT_OUT_ADD := 160;
   MachineConfig[4]."Unit Process"."EM - 201"."FCV201-1".CW.ENABLE := false;
   MachineConfig[4]."Unit Process"."EM - 201"."FIT201-1"."Type" := 0;
   MachineConfig[4]."Unit Process"."EM - 201"."FIT201-1".Address := 88;
   MachineConfig[4]."Unit Process"."EM - 201"."FIT201-1".Max := 10000.0;
   MachineConfig[4]."Unit Process"."EM - 201"."LA201-1".CW.ENABLE := False;
   MachineConfig[4]."Unit Process"."EM - 201"."PIT201-1".CW.ENABLE := true;
   MachineConfig[4]."Unit Process"."EM - 201"."PIT201-1".CW.EXIST := false;
   MachineConfig[4]."Unit Process"."EM - 22X"."AV220-1".CW.ENABLE := True;
   MachineConfig[4]."Unit Process"."EM - 22X"."AV220-1".CW.FB_CLS_EN := false;
   MachineConfig[4]."Unit Process"."EM - 22X"."AV220-1".CW.FB_OPN_EN := false;
   MachineConfig[4]."Unit Process"."EM - 22X"."AV220-1".CW.EXIST := False;
   MachineConfig[4]."Unit Process"."EM - 22X"."AV220-1".CW.VLV_W_FB := false;
   MachineConfig[4]."Unit Process"."EM - 22X"."AV220-1".FB_OPN_ADD := 8;
   MachineConfig[4]."Unit Process"."EM - 22X"."AV220-1".FB_CLS_ADD := 8;
   MachineConfig[4]."Unit Process"."EM - 22X"."AV220-1".ACT_OUT_ADD := 162;
   MachineConfig[4]."Unit Process"."EM - 22X"."AV460-1".CW.ENABLE := True;
   MachineConfig[4]."Unit Process"."EM - 22X"."AV460-1".CW.FB_CLS_EN := False;
   MachineConfig[4]."Unit Process"."EM - 22X"."AV460-1".CW.FB_OPN_EN := False;
   MachineConfig[4]."Unit Process"."EM - 22X"."AV460-1".CW.EXIST := False;
   MachineConfig[4]."Unit Process"."EM - 22X"."AV460-1".CW.VLV_W_FB := False;
   MachineConfig[4]."Unit Process"."EM - 22X"."AV460-1".FB_OPN_ADD := 8;
   MachineConfig[4]."Unit Process"."EM - 22X"."AV460-1".FB_CLS_ADD := 8;
   MachineConfig[4]."Unit Process"."EM - 22X"."AV460-1".ACT_OUT_ADD := 171;
   MachineConfig[4]."Unit Process"."EM - 22X"."FIT22X-1".CW.ENABLE := False;
   MachineConfig[4]."Unit Process"."EM - 22X"."PIT22X-1".CW.ENABLE := True;
   MachineConfig[4]."Unit Process"."EM - 22X"."PIT22X-1".CW.EXIST := false;
   MachineConfig[4]."Unit Process"."EM - 22X"."QT220-1".CW.ENABLE := True;
   MachineConfig[4]."Unit Process"."EM - 22X"."QT220-1".CW.EXIST := False;
   MachineConfig[4]."Unit Process"."EM - 22X"."PCV22X-1".CW.ENABLE := False;
   MachineConfig[4]."Unit Process"."EM - 340"."AV340-1".CW.ENABLE := True;
   MachineConfig[4]."Unit Process"."EM - 340"."AV340-1".CW.FB_CLS_EN := False;
   MachineConfig[4]."Unit Process"."EM - 340"."AV340-1".CW.FB_OPN_EN := False;
   MachineConfig[4]."Unit Process"."EM - 340"."AV340-1".CW.EXIST := False;
   MachineConfig[4]."Unit Process"."EM - 340"."AV340-1".CW.VLV_W_FB := False;
   MachineConfig[4]."Unit Process"."EM - 340"."AV340-1".FB_OPN_ADD := 8;
   MachineConfig[4]."Unit Process"."EM - 340"."AV340-1".FB_CLS_ADD := 8;
   MachineConfig[4]."Unit Process"."EM - 340"."AV340-1".ACT_OUT_ADD := 165;
   MachineConfig[4]."Unit Process"."EM - 340"."PIS340-1".Tag := 'PS301-1';
   MachineConfig[4]."Unit Dch"."EM - 222"."LS222-1".CW.ENABLE := False;
   MachineConfig[4]."Unit Dch"."EM - 222"."LS222-1".CW.EXIST := False;
   MachineConfig[4]."Unit Dch"."EM - 222"."P222-1".CW.EXIST := False;
   MachineConfig[4]."Unit Dch"."EM - 222"."P222-1".FB_RUN_ADD := 194;
   MachineConfig[4]."Unit Dch"."EM - 222"."P222-1".FB_RDY_ADD := 195;
   MachineConfig[4]."Unit Dch"."EM - 222"."P222-1".OUT_ACT_ADD := 182;
   MachineConfig[4]."Unit Dch"."EM - 222"."TS222-1".CW.ENABLE := False;
   MachineConfig[4]."Unit Dch"."EM - 300"."AV301-1".CW.ENABLE := True;
   MachineConfig[4]."Unit Dch"."EM - 300"."AV301-1".CW.FB_CLS_EN := false;
   MachineConfig[4]."Unit Dch"."EM - 300"."AV301-1".CW.FB_OPN_EN := false;
   MachineConfig[4]."Unit Dch"."EM - 300"."AV301-1".CW.VLV_W_FB := false;
   MachineConfig[4]."Unit Dch"."EM - 300"."AV301-1".FB_OPN_ADD := 8;
   MachineConfig[4]."Unit Dch"."EM - 300"."AV301-1".FB_CLS_ADD := 8;
   MachineConfig[4]."Unit Dch"."EM - 300"."AV301-1".ACT_OUT_ADD := 163;
   MachineConfig[4]."Unit Dch"."EM - 300"."AV320-1".CW.ENABLE := True;
   MachineConfig[4]."Unit Dch"."EM - 300"."AV320-1".CW.FB_CLS_EN := false;
   MachineConfig[4]."Unit Dch"."EM - 300"."AV320-1".CW.FB_OPN_EN := false;
   MachineConfig[4]."Unit Dch"."EM - 300"."AV320-1".CW.VLV_W_FB := false;
   MachineConfig[4]."Unit Dch"."EM - 300"."AV320-1".FB_OPN_ADD := 8;
   MachineConfig[4]."Unit Dch"."EM - 300"."AV320-1".FB_CLS_ADD := 8;
   MachineConfig[4]."Unit Dch"."EM - 300"."AV320-1".ACT_OUT_ADD := 164;
   MachineConfig[4]."Unit Dch"."EM - 375"."AV37X-1".CW.ENABLE := true;
   MachineConfig[4]."Unit Dch"."EM - 375"."AV37X-1".ACT_OUT_ADD := 166;
   MachineConfig[4]."Unit Dch"."EM - 375"."PIS375-1".CW.ENABLE := false;
   MachineConfig[4]."Unit Dch"."EM - 375"."PT37X-1".Tag := 'PT375-1';
   MachineConfig[4]."Unit Dch"."EM - 375"."PT37X-1".CW.ENABLE := true;
   MachineConfig[4]."Unit Dch"."EM - 375"."PT37X-1".Address := 76;
   MachineConfig[4]."Unit Dch"."EM - 375"."PT37X-1".Max := 600.0;
   MachineConfig[4]."Unit Dch"."EM - 506".IP506a.CW.ENABLE := True;
   MachineConfig[4]."Unit Dch"."EM - 506".AVDCH.TAG := '506b';
   MachineConfig[4]."Unit Dch"."EM - 506".AVDCH.CW.ENABLE := true;
   MachineConfig[4]."Unit Dch"."EM - 506".AVDCH.ACT_OUT_ADD := 167;
   MachineConfig[4].Options."EM - P201"."P201-1".FB_RUN_ADD := 196;
   MachineConfig[4].Options."EM - P201"."P201-1".FB_RDY_ADD := 197;
   MachineConfig[4].Options."EM - P201"."P201-1".OUT_ACT_ADD := 183;
   MachineConfig[4].Options."EM - P201"."P201-1".OUT_RST_ADD := 184;
   MachineConfig[4].Options."EM - P201"."P201-1_SPEED_REF".Address := 70;
   MachineConfig[5].Machine."Family" := 2;
   MachineConfig[5].Machine.TypeNo := 25;
   MachineConfig[5].Machine.Range := 2;
   MachineConfig[5].Machine.SepType := 1;
   MachineConfig[5].Machine.Frame := 1;
   MachineConfig[5].Machine.DchSystem := 2;
   MachineConfig[5].Machine.Spare_1 := 2;
   MachineConfig[5].Machine.FeedPump := 1;
   MachineConfig[5].Machine.Spare_2 := 2;
   MachineConfig[5].Machine.ConditionAlert := 1;
   MachineConfig[5].Machine.eWON := 1;
   MachineConfig[5]."Unit Sep"."EM - 100"."L-GREEN".CW.ENABLE := True;
   MachineConfig[5]."Unit Sep"."EM - 100"."L-GREEN".CW.EXIST := True;
   MachineConfig[5]."Unit Sep"."EM - 100"."L-YELLOW".Tag := 'L-BLUE';
   MachineConfig[5]."Unit Sep"."EM - 100".EMS.Address := 180;
   MachineConfig[5]."Unit Sep"."EM - 100".UPS.CW.ENABLE := True;
   MachineConfig[5]."Unit Sep"."EM - 100".UPS.CW.EXIST := True;
   MachineConfig[5]."Unit Sep"."EM - 100".UPS.Address := 181;
   MachineConfig[5]."Unit Sep"."EM - 100".EWON.CW.ENABLE := True;
   MachineConfig[5]."Unit Sep"."EM - 100".EWON.CW.EXIST := True;
   MachineConfig[5]."Unit Sep"."EM - 400"."AV409-1".CW.ENABLE := True;
   MachineConfig[5]."Unit Sep"."EM - 400"."AV409-1".ACT_OUT_ADD := 170;
   MachineConfig[5]."Unit Sep"."EM - 400"."FCV409-1".CW.ENABLE := True;
   MachineConfig[5]."Unit Sep"."EM - 400"."FIS409-1".CW.ENABLE := false;
   MachineConfig[5]."Unit Sep"."EM - 400"."FIT409-1".CW.ENABLE := True;
   MachineConfig[5]."Unit Sep"."EM - 400"."TT41X-1".CW.ENABLE := True;
   MachineConfig[5]."Unit Sep"."EM - 400"."TT41X-1"."Type" := 0;
   MachineConfig[5]."Unit Sep"."EM - 400"."TT41X-1".Address := 86;
   MachineConfig[5]."Unit Sep"."EM - 400"."TT41X-1".Min := -50.0;
   MachineConfig[5]."Unit Sep"."EM - 400"."TT41X-1".Max := 150.0;
   MachineConfig[5]."Unit Sep"."EM - 600"."AV63X/441-1".TAG := 'AV441-1';
   MachineConfig[5]."Unit Sep"."EM - 600"."AV63X/441-1".CW.ENABLE := True;
   MachineConfig[5]."Unit Sep"."EM - 600"."AV63X/441-1".CW.NO := False;
   MachineConfig[5]."Unit Sep"."EM - 600"."AV63X/441-1".CW.EXIST := True;
   MachineConfig[5]."Unit Sep"."EM - 600"."AV63X/441-1".ACT_OUT_ADD := 174;
   MachineConfig[5]."Unit Sep"."EM - 701".M701."TYPE" := 2;
   MachineConfig[5]."Unit Sep"."EM - 701".M701.FB_RUN_ADD := 8;
   MachineConfig[5]."Unit Sep"."EM - 701".M701.FB_RDY_ADD := 8;
   MachineConfig[5]."Unit Sep"."EM - 701".M701.OUT_ACT_ADD := 512;
   MachineConfig[5]."Unit Sep"."EM - 701".M701.OUT_RST_ADD := 8;
   MachineConfig[5]."Unit Sep"."EM - 730".TS730.CW.ENABLE := True;
   MachineConfig[5]."Unit Sep"."EM - 730".TS730.Address := 184;
   MachineConfig[5]."Unit Sep"."EM - 740"."P+F PS".Address := 180;
   MachineConfig[5]."Unit Sep"."EM - 740"."P+F OS".Address := 182;
   MachineConfig[5]."Unit Sep"."EM - 740"."P+F ERROR".Address := 183;
   MachineConfig[5]."Unit Sep"."EM - 750".YT75X.CW.ENABLE := True;
   MachineConfig[5]."Unit Sep"."EM - 750".YT75X.Address := 78;
   MachineConfig[5]."Unit Process"."EM - 201"."AV201-1".CW.ENABLE := True;
   MachineConfig[5]."Unit Process"."EM - 201"."AV201-1".CW.FB_CLS_EN := False;
   MachineConfig[5]."Unit Process"."EM - 201"."AV201-1".CW.FB_OPN_EN := False;
   MachineConfig[5]."Unit Process"."EM - 201"."AV201-1".CW.VLV_W_FB := False;
   MachineConfig[5]."Unit Process"."EM - 201"."AV201-1".FB_OPN_ADD := 8;
   MachineConfig[5]."Unit Process"."EM - 201"."AV201-1".FB_CLS_ADD := 8;
   MachineConfig[5]."Unit Process"."EM - 201"."AV201-1".ACT_OUT_ADD := 160;
   MachineConfig[5]."Unit Process"."EM - 201"."FCV201-1".CW.ENABLE := false;
   MachineConfig[5]."Unit Process"."EM - 201"."FIT201-1"."Type" := 0;
   MachineConfig[5]."Unit Process"."EM - 201"."FIT201-1".Address := 88;
   MachineConfig[5]."Unit Process"."EM - 201"."FIT201-1".Max := 50000.0;
   MachineConfig[5]."Unit Process"."EM - 201"."LA201-1".CW.ENABLE := False;
   MachineConfig[5]."Unit Process"."EM - 201"."PIT201-1".CW.ENABLE := true;
   MachineConfig[5]."Unit Process"."EM - 201"."PIT201-1".CW.EXIST := false;
   MachineConfig[5]."Unit Process"."EM - 22X"."AV220-1".CW.ENABLE := True;
   MachineConfig[5]."Unit Process"."EM - 22X"."AV220-1".CW.FB_CLS_EN := false;
   MachineConfig[5]."Unit Process"."EM - 22X"."AV220-1".CW.FB_OPN_EN := false;
   MachineConfig[5]."Unit Process"."EM - 22X"."AV220-1".CW.VLV_W_FB := false;
   MachineConfig[5]."Unit Process"."EM - 22X"."AV220-1".FB_OPN_ADD := 8;
   MachineConfig[5]."Unit Process"."EM - 22X"."AV220-1".FB_CLS_ADD := 8;
   MachineConfig[5]."Unit Process"."EM - 22X"."AV220-1".ACT_OUT_ADD := 162;
   MachineConfig[5]."Unit Process"."EM - 22X"."AV460-1".CW.ENABLE := True;
   MachineConfig[5]."Unit Process"."EM - 22X"."AV460-1".CW.FB_CLS_EN := false;
   MachineConfig[5]."Unit Process"."EM - 22X"."AV460-1".CW.FB_OPN_EN := false;
   MachineConfig[5]."Unit Process"."EM - 22X"."AV460-1".CW.VLV_W_FB := False;
   MachineConfig[5]."Unit Process"."EM - 22X"."AV460-1".FB_OPN_ADD := 8;
   MachineConfig[5]."Unit Process"."EM - 22X"."AV460-1".FB_CLS_ADD := 8;
   MachineConfig[5]."Unit Process"."EM - 22X"."AV460-1".ACT_OUT_ADD := 171;
   MachineConfig[5]."Unit Process"."EM - 22X"."FIT22X-1".CW.ENABLE := False;
   MachineConfig[5]."Unit Process"."EM - 22X"."PIT22X-1".CW.ENABLE := True;
   MachineConfig[5]."Unit Process"."EM - 22X"."PIT22X-1".CW.EXIST := false;
   MachineConfig[5]."Unit Process"."EM - 22X"."QT220-1".CW.ENABLE := True;
   MachineConfig[5]."Unit Process"."EM - 22X"."QT220-1".CW.EXIST := False;
   MachineConfig[5]."Unit Process"."EM - 22X"."PCV22X-1".CW.ENABLE := False;
   MachineConfig[5]."Unit Process"."EM - 340"."AV340-1".CW.ENABLE := True;
   MachineConfig[5]."Unit Process"."EM - 340"."AV340-1".CW.FB_CLS_EN := False;
   MachineConfig[5]."Unit Process"."EM - 340"."AV340-1".CW.FB_OPN_EN := False;
   MachineConfig[5]."Unit Process"."EM - 340"."AV340-1".CW.VLV_W_FB := False;
   MachineConfig[5]."Unit Process"."EM - 340"."AV340-1".FB_OPN_ADD := 8;
   MachineConfig[5]."Unit Process"."EM - 340"."AV340-1".FB_CLS_ADD := 8;
   MachineConfig[5]."Unit Process"."EM - 340"."AV340-1".ACT_OUT_ADD := 165;
   MachineConfig[5]."Unit Dch"."EM - 222"."LS222-1".CW.EXIST := False;
   MachineConfig[5]."Unit Dch"."EM - 222"."P222-1".CW.EXIST := False;
   MachineConfig[5]."Unit Dch"."EM - 222"."P222-1".FB_RUN_ADD := 194;
   MachineConfig[5]."Unit Dch"."EM - 222"."P222-1".FB_RDY_ADD := 195;
   MachineConfig[5]."Unit Dch"."EM - 222"."P222-1".OUT_ACT_ADD := 182;
   MachineConfig[5]."Unit Dch"."EM - 222"."TS222-1".CW.ENABLE := False;
   MachineConfig[5]."Unit Dch"."EM - 300"."AV301-1".CW.ENABLE := True;
   MachineConfig[5]."Unit Dch"."EM - 300"."AV301-1".CW.FB_CLS_EN := false;
   MachineConfig[5]."Unit Dch"."EM - 300"."AV301-1".CW.FB_OPN_EN := false;
   MachineConfig[5]."Unit Dch"."EM - 300"."AV301-1".CW.VLV_W_FB := false;
   MachineConfig[5]."Unit Dch"."EM - 300"."AV301-1".FB_OPN_ADD := 8;
   MachineConfig[5]."Unit Dch"."EM - 300"."AV301-1".FB_CLS_ADD := 8;
   MachineConfig[5]."Unit Dch"."EM - 300"."AV301-1".ACT_OUT_ADD := 163;
   MachineConfig[5]."Unit Dch"."EM - 300"."AV304-1".TAG := 'AV301-1';
   MachineConfig[5]."Unit Dch"."EM - 300"."AV304-1".ACT_OUT_ADD := 163;
   MachineConfig[5]."Unit Dch"."EM - 300"."AV320-1".CW.ENABLE := true;
   MachineConfig[5]."Unit Dch"."EM - 300"."AV320-1".CW.FB_CLS_EN := false;
   MachineConfig[5]."Unit Dch"."EM - 300"."AV320-1".CW.FB_OPN_EN := false;
   MachineConfig[5]."Unit Dch"."EM - 300"."AV320-1".CW.VLV_W_FB := false;
   MachineConfig[5]."Unit Dch"."EM - 300"."AV320-1".FB_OPN_ADD := 8;
   MachineConfig[5]."Unit Dch"."EM - 300"."AV320-1".FB_CLS_ADD := 8;
   MachineConfig[5]."Unit Dch"."EM - 300"."AV320-1".ACT_OUT_ADD := 164;
   MachineConfig[5]."Unit Dch"."EM - 300"."AV635-1".ACT_OUT_ADD := 174;
   MachineConfig[5]."Unit Dch"."EM - 375"."AV37X-1".CW.ENABLE := true;
   MachineConfig[5]."Unit Dch"."EM - 375"."AV37X-1".ACT_OUT_ADD := 166;
   MachineConfig[5]."Unit Dch"."EM - 375"."PIS375-1".CW.ENABLE := false;
   MachineConfig[5]."Unit Dch"."EM - 375"."PT37X-1".Tag := 'PT375-1';
   MachineConfig[5]."Unit Dch"."EM - 375"."PT37X-1".CW.ENABLE := True;
   MachineConfig[5]."Unit Dch"."EM - 375"."PT37X-1".Address := 76;
   MachineConfig[5]."Unit Dch"."EM - 375"."PT37X-1".Max := 600.0;
   MachineConfig[5]."Unit Dch"."EM - 506".IP506a.CW.ENABLE := True;
   MachineConfig[5]."Unit Dch"."EM - 506".AVDCH.TAG := '506b';
   MachineConfig[5]."Unit Dch"."EM - 506".AVDCH.CW.ENABLE := true;
   MachineConfig[5]."Unit Dch"."EM - 506".AVDCH.ACT_OUT_ADD := 167;
   MachineConfig[5].Options."EM - P201"."P201-1".FB_RUN_ADD := 196;
   MachineConfig[5].Options."EM - P201"."P201-1".FB_RDY_ADD := 197;
   MachineConfig[5].Options."EM - P201"."P201-1".OUT_ACT_ADD := 183;
   MachineConfig[5].Options."EM - P201"."P201-1".OUT_RST_ADD := 184;
   MachineConfig[6].Machine."Family" := 2;
   MachineConfig[6].Machine.TypeNo := 26;
   MachineConfig[6].Machine.Range := 2;
   MachineConfig[6].Machine.SepType := 1;
   MachineConfig[6].Machine.Frame := 1;
   MachineConfig[6].Machine.DchSystem := 2;
   MachineConfig[6].Machine.Spare_1 := 2;
   MachineConfig[6].Machine.FeedPump := 1;
   MachineConfig[6].Machine.Spare_2 := 2;
   MachineConfig[6].Machine.ConditionAlert := 1;
   MachineConfig[6].Machine.eWON := 1;
   MachineConfig[6]."Unit Sep"."EM - 100"."L-GREEN".CW.ENABLE := True;
   MachineConfig[6]."Unit Sep"."EM - 100"."L-GREEN".CW.EXIST := True;
   MachineConfig[6]."Unit Sep"."EM - 100"."L-YELLOW".Tag := 'L-BLUE';
   MachineConfig[6]."Unit Sep"."EM - 100".EMS.Address := 180;
   MachineConfig[6]."Unit Sep"."EM - 100".UPS.CW.ENABLE := True;
   MachineConfig[6]."Unit Sep"."EM - 100".UPS.CW.EXIST := True;
   MachineConfig[6]."Unit Sep"."EM - 100".UPS.Address := 181;
   MachineConfig[6]."Unit Sep"."EM - 100".EWON.CW.ENABLE := True;
   MachineConfig[6]."Unit Sep"."EM - 100".EWON.CW.EXIST := True;
   MachineConfig[6]."Unit Sep"."EM - 400"."AV409-1".CW.ENABLE := True;
   MachineConfig[6]."Unit Sep"."EM - 400"."AV409-1".ACT_OUT_ADD := 170;
   MachineConfig[6]."Unit Sep"."EM - 400"."FCV409-1".CW.ENABLE := True;
   MachineConfig[6]."Unit Sep"."EM - 400"."FIS409-1".CW.ENABLE := false;
   MachineConfig[6]."Unit Sep"."EM - 400"."FIT409-1".CW.ENABLE := True;
   MachineConfig[6]."Unit Sep"."EM - 400"."TT41X-1".CW.ENABLE := True;
   MachineConfig[6]."Unit Sep"."EM - 400"."TT41X-1"."Type" := 0;
   MachineConfig[6]."Unit Sep"."EM - 400"."TT41X-1".Address := 86;
   MachineConfig[6]."Unit Sep"."EM - 400"."TT41X-1".Min := -50.0;
   MachineConfig[6]."Unit Sep"."EM - 400"."TT41X-1".Max := 150.0;
   MachineConfig[6]."Unit Sep"."EM - 600"."AV615-1".ACT_OUT_ADD := 173;
   MachineConfig[6]."Unit Sep"."EM - 600"."AV63X/441-1".TAG := 'AV635-1';
   MachineConfig[6]."Unit Sep"."EM - 600"."AV63X/441-1".CW.ENABLE := True;
   MachineConfig[6]."Unit Sep"."EM - 600"."AV63X/441-1".CW.NO := True;
   MachineConfig[6]."Unit Sep"."EM - 600"."AV63X/441-1".CW.EXIST := True;
   MachineConfig[6]."Unit Sep"."EM - 600"."AV63X/441-1".ACT_OUT_ADD := 174;
   MachineConfig[6]."Unit Sep"."EM - 600"."FIS635-1".Tag := 'FIS635-1';
   MachineConfig[6]."Unit Sep"."EM - 600"."FIS635-1".CW.ENABLE := True;
   MachineConfig[6]."Unit Sep"."EM - 701".M701."TYPE" := 2;
   MachineConfig[6]."Unit Sep"."EM - 701".M701.FB_RUN_ADD := 8;
   MachineConfig[6]."Unit Sep"."EM - 701".M701.FB_RDY_ADD := 8;
   MachineConfig[6]."Unit Sep"."EM - 701".M701.OUT_ACT_ADD := 512;
   MachineConfig[6]."Unit Sep"."EM - 701".M701.OUT_RST_ADD := 8;
   MachineConfig[6]."Unit Sep"."EM - 730".TS730.CW.ENABLE := True;
   MachineConfig[6]."Unit Sep"."EM - 730".TS730.Address := 184;
   MachineConfig[6]."Unit Sep"."EM - 740"."P+F PS".Address := 180;
   MachineConfig[6]."Unit Sep"."EM - 740"."P+F OS".Address := 182;
   MachineConfig[6]."Unit Sep"."EM - 740"."P+F ERROR".Address := 183;
   MachineConfig[6]."Unit Sep"."EM - 750".YT75X.CW.ENABLE := True;
   MachineConfig[6]."Unit Sep"."EM - 750".YT75X.Address := 78;
   MachineConfig[6]."Unit Process"."EM - 201"."AV201-1".CW.ENABLE := True;
   MachineConfig[6]."Unit Process"."EM - 201"."AV201-1".CW.FB_CLS_EN := False;
   MachineConfig[6]."Unit Process"."EM - 201"."AV201-1".CW.FB_OPN_EN := False;
   MachineConfig[6]."Unit Process"."EM - 201"."AV201-1".CW.VLV_W_FB := False;
   MachineConfig[6]."Unit Process"."EM - 201"."AV201-1".FB_OPN_ADD := 8;
   MachineConfig[6]."Unit Process"."EM - 201"."AV201-1".FB_CLS_ADD := 8;
   MachineConfig[6]."Unit Process"."EM - 201"."AV201-1".ACT_OUT_ADD := 160;
   MachineConfig[6]."Unit Process"."EM - 201"."FCV201-1".CW.ENABLE := false;
   MachineConfig[6]."Unit Process"."EM - 201"."FIT201-1"."Type" := 0;
   MachineConfig[6]."Unit Process"."EM - 201"."FIT201-1".Address := 88;
   MachineConfig[6]."Unit Process"."EM - 201"."FIT201-1".Max := 40000.0;
   MachineConfig[6]."Unit Process"."EM - 201"."LA201-1".CW.ENABLE := False;
   MachineConfig[6]."Unit Process"."EM - 201"."PIT201-1".CW.EXIST := False;
   MachineConfig[6]."Unit Process"."EM - 22X"."AV220-1".TAG := 'AV220-1';
   MachineConfig[6]."Unit Process"."EM - 22X"."AV220-1".CW.ENABLE := True;
   MachineConfig[6]."Unit Process"."EM - 22X"."AV220-1".CW.FB_CLS_EN := False;
   MachineConfig[6]."Unit Process"."EM - 22X"."AV220-1".CW.FB_OPN_EN := False;
   MachineConfig[6]."Unit Process"."EM - 22X"."AV220-1".CW.VLV_W_FB := False;
   MachineConfig[6]."Unit Process"."EM - 22X"."AV220-1".FB_OPN_ADD := 8;
   MachineConfig[6]."Unit Process"."EM - 22X"."AV220-1".FB_CLS_ADD := 8;
   MachineConfig[6]."Unit Process"."EM - 22X"."AV220-1".ACT_OUT_ADD := 162;
   MachineConfig[6]."Unit Process"."EM - 22X"."AV460-1".CW.ENABLE := True;
   MachineConfig[6]."Unit Process"."EM - 22X"."AV460-1".CW.FB_CLS_EN := false;
   MachineConfig[6]."Unit Process"."EM - 22X"."AV460-1".CW.FB_OPN_EN := false;
   MachineConfig[6]."Unit Process"."EM - 22X"."AV460-1".CW.VLV_W_FB := False;
   MachineConfig[6]."Unit Process"."EM - 22X"."AV460-1".FB_OPN_ADD := 8;
   MachineConfig[6]."Unit Process"."EM - 22X"."AV460-1".FB_CLS_ADD := 8;
   MachineConfig[6]."Unit Process"."EM - 22X"."AV460-1".ACT_OUT_ADD := 171;
   MachineConfig[6]."Unit Process"."EM - 22X"."FIT22X-1".CW.ENABLE := False;
   MachineConfig[6]."Unit Process"."EM - 22X"."PIT22X-1".CW.ENABLE := True;
   MachineConfig[6]."Unit Process"."EM - 22X"."PIT22X-1".CW.EXIST := False;
   MachineConfig[6]."Unit Process"."EM - 22X"."QT220-1".CW.ENABLE := True;
   MachineConfig[6]."Unit Process"."EM - 22X"."QT220-1".CW.EXIST := False;
   MachineConfig[6]."Unit Process"."EM - 22X"."PCV22X-1".CW.ENABLE := False;
   MachineConfig[6]."Unit Process"."EM - 340"."AV340-1".CW.ENABLE := True;
   MachineConfig[6]."Unit Process"."EM - 340"."AV340-1".CW.FB_CLS_EN := False;
   MachineConfig[6]."Unit Process"."EM - 340"."AV340-1".CW.FB_OPN_EN := False;
   MachineConfig[6]."Unit Process"."EM - 340"."AV340-1".CW.VLV_W_FB := False;
   MachineConfig[6]."Unit Process"."EM - 340"."AV340-1".FB_OPN_ADD := 8;
   MachineConfig[6]."Unit Process"."EM - 340"."AV340-1".FB_CLS_ADD := 8;
   MachineConfig[6]."Unit Process"."EM - 340"."AV340-1".ACT_OUT_ADD := 165;
   MachineConfig[6]."Unit Process"."EM - 340"."PIS340-1".Tag := 'PS301-1';
   MachineConfig[6]."Unit Dch"."EM - 222"."LS222-1".CW.ENABLE := False;
   MachineConfig[6]."Unit Dch"."EM - 222"."LS222-1".CW.EXIST := False;
   MachineConfig[6]."Unit Dch"."EM - 222"."P222-1".CW.EXIST := False;
   MachineConfig[6]."Unit Dch"."EM - 222"."P222-1".FB_RUN_ADD := 194;
   MachineConfig[6]."Unit Dch"."EM - 222"."P222-1".FB_RDY_ADD := 195;
   MachineConfig[6]."Unit Dch"."EM - 222"."P222-1".OUT_ACT_ADD := 182;
   MachineConfig[6]."Unit Dch"."EM - 222"."TS222-1".CW.ENABLE := False;
   MachineConfig[6]."Unit Dch"."EM - 300"."AV301-1".CW.FB_CLS_EN := False;
   MachineConfig[6]."Unit Dch"."EM - 300"."AV301-1".CW.FB_OPN_EN := False;
   MachineConfig[6]."Unit Dch"."EM - 300"."AV301-1".CW.VLV_W_FB := False;
   MachineConfig[6]."Unit Dch"."EM - 300"."AV301-1".FB_OPN_ADD := 8;
   MachineConfig[6]."Unit Dch"."EM - 300"."AV301-1".FB_CLS_ADD := 8;
   MachineConfig[6]."Unit Dch"."EM - 300"."AV301-1".ACT_OUT_ADD := 163;
   MachineConfig[6]."Unit Dch"."EM - 300"."AV304-1".TAG := 'AV301-1';
   MachineConfig[6]."Unit Dch"."EM - 300"."AV304-1".ACT_OUT_ADD := 163;
   MachineConfig[6]."Unit Dch"."EM - 300"."AV320-1".CW.ENABLE := true;
   MachineConfig[6]."Unit Dch"."EM - 300"."AV320-1".CW.FB_CLS_EN := false;
   MachineConfig[6]."Unit Dch"."EM - 300"."AV320-1".CW.FB_OPN_EN := false;
   MachineConfig[6]."Unit Dch"."EM - 300"."AV320-1".CW.VLV_W_FB := false;
   MachineConfig[6]."Unit Dch"."EM - 300"."AV320-1".FB_OPN_ADD := 8;
   MachineConfig[6]."Unit Dch"."EM - 300"."AV320-1".FB_CLS_ADD := 8;
   MachineConfig[6]."Unit Dch"."EM - 300"."AV320-1".ACT_OUT_ADD := 164;
   MachineConfig[6]."Unit Dch"."EM - 300"."AV635-1".ACT_OUT_ADD := 174;
   MachineConfig[6]."Unit Dch"."EM - 375"."AV37X-1".CW.ENABLE := true;
   MachineConfig[6]."Unit Dch"."EM - 375"."AV37X-1".ACT_OUT_ADD := 166;
   MachineConfig[6]."Unit Dch"."EM - 375"."PIS375-1".CW.ENABLE := false;
   MachineConfig[6]."Unit Dch"."EM - 375"."PT37X-1".Tag := 'PT375-1';
   MachineConfig[6]."Unit Dch"."EM - 375"."PT37X-1".CW.ENABLE := true;
   MachineConfig[6]."Unit Dch"."EM - 375"."PT37X-1".Address := 76;
   MachineConfig[6]."Unit Dch"."EM - 375"."PT37X-1".Max := 600.0;
   MachineConfig[6]."Unit Dch"."EM - 506".IP506a.CW.ENABLE := True;
   MachineConfig[6]."Unit Dch"."EM - 506".AVDCH.TAG := '506b';
   MachineConfig[6]."Unit Dch"."EM - 506".AVDCH.CW.ENABLE := true;
   MachineConfig[6]."Unit Dch"."EM - 506".AVDCH.ACT_OUT_ADD := 167;
   MachineConfig[6].Options."EM - P201"."P201-1".FB_RUN_ADD := 196;
   MachineConfig[6].Options."EM - P201"."P201-1".FB_RDY_ADD := 197;
   MachineConfig[6].Options."EM - P201"."P201-1".OUT_ACT_ADD := 183;
   MachineConfig[6].Options."EM - P201"."P201-1".OUT_RST_ADD := 184;
   MachineConfig[6].Options."EM - P201"."P201-1_SPEED_REF".Address := 70;
   MachineConfig[7].Machine."Family" := 2;
   MachineConfig[7].Machine.TypeNo := 27;
   MachineConfig[7].Machine.Range := 2;
   MachineConfig[7].Machine.SepType := 1;
   MachineConfig[7].Machine.Frame := 1;
   MachineConfig[7].Machine.DchSystem := 2;
   MachineConfig[7].Machine.Spare_1 := 2;
   MachineConfig[7].Machine.FeedPump := 1;
   MachineConfig[7].Machine.Spare_2 := 2;
   MachineConfig[7].Machine.ConditionAlert := 1;
   MachineConfig[7].Machine.eWON := 1;
   MachineConfig[7]."Unit Sep"."EM - 100"."L-GREEN".CW.ENABLE := True;
   MachineConfig[7]."Unit Sep"."EM - 100"."L-GREEN".CW.EXIST := True;
   MachineConfig[7]."Unit Sep"."EM - 100"."L-YELLOW".Tag := 'L-BLUE';
   MachineConfig[7]."Unit Sep"."EM - 100".EMS.Address := 180;
   MachineConfig[7]."Unit Sep"."EM - 100".UPS.CW.ENABLE := True;
   MachineConfig[7]."Unit Sep"."EM - 100".UPS.CW.EXIST := True;
   MachineConfig[7]."Unit Sep"."EM - 100".UPS.Address := 181;
   MachineConfig[7]."Unit Sep"."EM - 100".EWON.CW.ENABLE := True;
   MachineConfig[7]."Unit Sep"."EM - 100".EWON.CW.EXIST := True;
   MachineConfig[7]."Unit Sep"."EM - 400"."AV409-1".CW.ENABLE := True;
   MachineConfig[7]."Unit Sep"."EM - 400"."AV409-1".ACT_OUT_ADD := 170;
   MachineConfig[7]."Unit Sep"."EM - 400"."FCV409-1".CW.ENABLE := True;
   MachineConfig[7]."Unit Sep"."EM - 400"."FIS409-1".CW.ENABLE := False;
   MachineConfig[7]."Unit Sep"."EM - 400"."FIT409-1".CW.ENABLE := True;
   MachineConfig[7]."Unit Sep"."EM - 400"."TT41X-1".CW.ENABLE := True;
   MachineConfig[7]."Unit Sep"."EM - 400"."TT41X-1"."Type" := 0;
   MachineConfig[7]."Unit Sep"."EM - 400"."TT41X-1".Address := 86;
   MachineConfig[7]."Unit Sep"."EM - 400"."TT41X-1".Min := -50.0;
   MachineConfig[7]."Unit Sep"."EM - 400"."TT41X-1".Max := 150.0;
   MachineConfig[7]."Unit Sep"."EM - 600"."AV615-1".CW.ENABLE := True;
   MachineConfig[7]."Unit Sep"."EM - 600"."AV615-1".CW.NO := True;
   MachineConfig[7]."Unit Sep"."EM - 600"."AV615-1".CW.EXIST := True;
   MachineConfig[7]."Unit Sep"."EM - 600"."AV615-1".ACT_OUT_ADD := 173;
   MachineConfig[7]."Unit Sep"."EM - 600"."AV63X/441-1".TAG := 'AV635-1';
   MachineConfig[7]."Unit Sep"."EM - 600"."AV63X/441-1".CW.ENABLE := True;
   MachineConfig[7]."Unit Sep"."EM - 600"."AV63X/441-1".CW.NO := True;
   MachineConfig[7]."Unit Sep"."EM - 600"."AV63X/441-1".CW.EXIST := True;
   MachineConfig[7]."Unit Sep"."EM - 600"."AV63X/441-1".ACT_OUT_ADD := 174;
   MachineConfig[7]."Unit Sep"."EM - 600"."FIS615-1".CW.ENABLE := True;
   MachineConfig[7]."Unit Sep"."EM - 600"."FIS635-1".CW.ENABLE := True;
   MachineConfig[7]."Unit Sep"."EM - 701".M701."TYPE" := 2;
   MachineConfig[7]."Unit Sep"."EM - 701".M701.FB_RUN_ADD := 8;
   MachineConfig[7]."Unit Sep"."EM - 701".M701.FB_RDY_ADD := 8;
   MachineConfig[7]."Unit Sep"."EM - 701".M701.OUT_ACT_ADD := 512;
   MachineConfig[7]."Unit Sep"."EM - 701".M701.OUT_RST_ADD := 8;
   MachineConfig[7]."Unit Sep"."EM - 730".TS730.CW.ENABLE := True;
   MachineConfig[7]."Unit Sep"."EM - 730".TS730.Address := 184;
   MachineConfig[7]."Unit Sep"."EM - 740"."P+F PS".Address := 180;
   MachineConfig[7]."Unit Sep"."EM - 740"."P+F OS".Address := 182;
   MachineConfig[7]."Unit Sep"."EM - 740"."P+F ERROR".Address := 183;
   MachineConfig[7]."Unit Sep"."EM - 750".YT75X.Address := 78;
   MachineConfig[7]."Unit Process"."EM - 201"."AV201-1".CW.ENABLE := True;
   MachineConfig[7]."Unit Process"."EM - 201"."AV201-1".CW.FB_CLS_EN := False;
   MachineConfig[7]."Unit Process"."EM - 201"."AV201-1".CW.FB_OPN_EN := False;
   MachineConfig[7]."Unit Process"."EM - 201"."AV201-1".CW.VLV_W_FB := False;
   MachineConfig[7]."Unit Process"."EM - 201"."AV201-1".FB_OPN_ADD := 8;
   MachineConfig[7]."Unit Process"."EM - 201"."AV201-1".FB_CLS_ADD := 8;
   MachineConfig[7]."Unit Process"."EM - 201"."AV201-1".ACT_OUT_ADD := 160;
   MachineConfig[7]."Unit Process"."EM - 201"."AV460a-1".CW.ENABLE := True;
   MachineConfig[7]."Unit Process"."EM - 201"."FCV201-1".CW.ENABLE := False;
   MachineConfig[7]."Unit Process"."EM - 201"."FIT201-1"."Type" := 0;
   MachineConfig[7]."Unit Process"."EM - 201"."FIT201-1".Address := 88;
   MachineConfig[7]."Unit Process"."EM - 201"."FIT201-1".Max := 50000.0;
   MachineConfig[7]."Unit Process"."EM - 201"."LA201-1".CW.ENABLE := False;
   MachineConfig[7]."Unit Process"."EM - 201"."PIT201-1".CW.ENABLE := True;
   MachineConfig[7]."Unit Process"."EM - 201"."PIT201-1".CW.EXIST := False;
   MachineConfig[7]."Unit Process"."EM - 22X"."AV220-1".CW.ENABLE := True;
   MachineConfig[7]."Unit Process"."EM - 22X"."AV220-1".CW.FB_CLS_EN := False;
   MachineConfig[7]."Unit Process"."EM - 22X"."AV220-1".CW.FB_OPN_EN := False;
   MachineConfig[7]."Unit Process"."EM - 22X"."AV220-1".CW.VLV_W_FB := False;
   MachineConfig[7]."Unit Process"."EM - 22X"."AV220-1".FB_OPN_ADD := 8;
   MachineConfig[7]."Unit Process"."EM - 22X"."AV220-1".FB_CLS_ADD := 8;
   MachineConfig[7]."Unit Process"."EM - 22X"."AV220-1".ACT_OUT_ADD := 162;
   MachineConfig[7]."Unit Process"."EM - 22X"."AV460-1".CW.ENABLE := True;
   MachineConfig[7]."Unit Process"."EM - 22X"."AV460-1".CW.FB_CLS_EN := False;
   MachineConfig[7]."Unit Process"."EM - 22X"."AV460-1".CW.FB_OPN_EN := False;
   MachineConfig[7]."Unit Process"."EM - 22X"."AV460-1".CW.VLV_W_FB := False;
   MachineConfig[7]."Unit Process"."EM - 22X"."AV460-1".FB_OPN_ADD := 8;
   MachineConfig[7]."Unit Process"."EM - 22X"."AV460-1".FB_CLS_ADD := 8;
   MachineConfig[7]."Unit Process"."EM - 22X"."AV460-1".ACT_OUT_ADD := 171;
   MachineConfig[7]."Unit Process"."EM - 22X"."FIT22X-1".CW.ENABLE := False;
   MachineConfig[7]."Unit Process"."EM - 22X"."PIT22X-1".CW.ENABLE := True;
   MachineConfig[7]."Unit Process"."EM - 22X"."PIT22X-1".CW.EXIST := False;
   MachineConfig[7]."Unit Process"."EM - 22X"."QT220-1".CW.ENABLE := True;
   MachineConfig[7]."Unit Process"."EM - 22X"."QT220-1".CW.EXIST := False;
   MachineConfig[7]."Unit Process"."EM - 22X"."PCV22X-1".CW.ENABLE := False;
   MachineConfig[7]."Unit Process"."EM - 340"."AV340-1".CW.ENABLE := True;
   MachineConfig[7]."Unit Process"."EM - 340"."AV340-1".CW.FB_CLS_EN := False;
   MachineConfig[7]."Unit Process"."EM - 340"."AV340-1".CW.FB_OPN_EN := False;
   MachineConfig[7]."Unit Process"."EM - 340"."AV340-1".CW.VLV_W_FB := False;
   MachineConfig[7]."Unit Process"."EM - 340"."AV340-1".FB_OPN_ADD := 8;
   MachineConfig[7]."Unit Process"."EM - 340"."AV340-1".FB_CLS_ADD := 8;
   MachineConfig[7]."Unit Process"."EM - 340"."AV340-1".ACT_OUT_ADD := 165;
   MachineConfig[7]."Unit Process"."EM - 340"."V340-1".CW.ENABLE := True;
   MachineConfig[7]."Unit Process"."EM - 340"."V340-1".Address := 170;
   MachineConfig[7]."Unit Dch"."EM - 222"."LS222-1".CW.ENABLE := False;
   MachineConfig[7]."Unit Dch"."EM - 222"."P222-1".CW.ENABLE := True;
   MachineConfig[7]."Unit Dch"."EM - 222"."P222-1".CW.EXIST := False;
   MachineConfig[7]."Unit Dch"."EM - 222"."P222-1".FB_RUN_ADD := 194;
   MachineConfig[7]."Unit Dch"."EM - 222"."P222-1".FB_RDY_ADD := 195;
   MachineConfig[7]."Unit Dch"."EM - 222"."P222-1".OUT_ACT_ADD := 182;
   MachineConfig[7]."Unit Dch"."EM - 222"."TS222-1".CW.ENABLE := False;
   MachineConfig[7]."Unit Dch"."EM - 300"."AV301-1".CW.ENABLE := True;
   MachineConfig[7]."Unit Dch"."EM - 300"."AV301-1".CW.FB_CLS_EN := False;
   MachineConfig[7]."Unit Dch"."EM - 300"."AV301-1".CW.FB_OPN_EN := False;
   MachineConfig[7]."Unit Dch"."EM - 300"."AV301-1".CW.VLV_W_FB := False;
   MachineConfig[7]."Unit Dch"."EM - 300"."AV301-1".FB_OPN_ADD := 8;
   MachineConfig[7]."Unit Dch"."EM - 300"."AV301-1".FB_CLS_ADD := 8;
   MachineConfig[7]."Unit Dch"."EM - 300"."AV301-1".ACT_OUT_ADD := 163;
   MachineConfig[7]."Unit Dch"."EM - 300"."AV320-1".CW.ENABLE := True;
   MachineConfig[7]."Unit Dch"."EM - 300"."AV320-1".CW.FB_CLS_EN := False;
   MachineConfig[7]."Unit Dch"."EM - 300"."AV320-1".CW.FB_OPN_EN := False;
   MachineConfig[7]."Unit Dch"."EM - 300"."AV320-1".CW.VLV_W_FB := False;
   MachineConfig[7]."Unit Dch"."EM - 300"."AV320-1".FB_OPN_ADD := 8;
   MachineConfig[7]."Unit Dch"."EM - 300"."AV320-1".FB_CLS_ADD := 8;
   MachineConfig[7]."Unit Dch"."EM - 300"."AV320-1".ACT_OUT_ADD := 164;
   MachineConfig[7]."Unit Dch"."EM - 300"."AV635-1".TAG := 'AV635a-1';
   MachineConfig[7]."Unit Dch"."EM - 375"."AV37X-1".CW.ENABLE := True;
   MachineConfig[7]."Unit Dch"."EM - 375"."AV37X-1".ACT_OUT_ADD := 166;
   MachineConfig[7]."Unit Dch"."EM - 375"."PIS375-1".CW.ENABLE := False;
   MachineConfig[7]."Unit Dch"."EM - 375"."PT37X-1".Tag := 'PT375-1';
   MachineConfig[7]."Unit Dch"."EM - 375"."PT37X-1".CW.ENABLE := True;
   MachineConfig[7]."Unit Dch"."EM - 375"."PT37X-1".Address := 76;
   MachineConfig[7]."Unit Dch"."EM - 375"."PT37X-1".Max := 600.0;
   MachineConfig[7]."Unit Dch"."EM - 506".IP506a.CW.ENABLE := True;
   MachineConfig[7]."Unit Dch"."EM - 506".AVDCH.TAG := '506b';
   MachineConfig[7]."Unit Dch"."EM - 506".AVDCH.CW.ENABLE := True;
   MachineConfig[7]."Unit Dch"."EM - 506".AVDCH.ACT_OUT_ADD := 167;
   MachineConfig[7].Options."EM - P201"."P201-1".FB_RUN_ADD := 196;
   MachineConfig[7].Options."EM - P201"."P201-1".FB_RDY_ADD := 197;
   MachineConfig[7].Options."EM - P201"."P201-1".OUT_ACT_ADD := 183;
   MachineConfig[7].Options."EM - P201"."P201-1".OUT_RST_ADD := 184;
   MachineConfig[7].Options."EM - P201"."P201-1_SPEED_REF".Address := 70;
   MachineConfig[8].Machine."Family" := 2;
   MachineConfig[8].Machine.TypeNo := 28;
   MachineConfig[8].Machine.Range := 2;
   MachineConfig[8].Machine.SepType := 1;
   MachineConfig[8].Machine.Frame := 1;
   MachineConfig[8].Machine.DchSystem := 2;
   MachineConfig[8].Machine.Spare_1 := 2;
   MachineConfig[8].Machine.FeedPump := 1;
   MachineConfig[8].Machine.Spare_2 := 2;
   MachineConfig[8].Machine.ConditionAlert := 1;
   MachineConfig[8].Machine.eWON := 1;
   MachineConfig[8]."Unit Sep"."EM - 100"."L-GREEN".CW.ENABLE := True;
   MachineConfig[8]."Unit Sep"."EM - 100"."L-GREEN".CW.EXIST := True;
   MachineConfig[8]."Unit Sep"."EM - 100"."L-YELLOW".Tag := 'L-BLUE';
   MachineConfig[8]."Unit Sep"."EM - 100"."L-RED".CW.ENABLE := True;
   MachineConfig[8]."Unit Sep"."EM - 100"."L-RED".CW.EXIST := True;
   MachineConfig[8]."Unit Sep"."EM - 100".EMS.Address := 180;
   MachineConfig[8]."Unit Sep"."EM - 100".UPS.CW.ENABLE := True;
   MachineConfig[8]."Unit Sep"."EM - 100".UPS.CW.EXIST := True;
   MachineConfig[8]."Unit Sep"."EM - 100".UPS.Address := 181;
   MachineConfig[8]."Unit Sep"."EM - 100".EWON.CW.ENABLE := True;
   MachineConfig[8]."Unit Sep"."EM - 100".EWON.CW.EXIST := True;
   MachineConfig[8]."Unit Sep"."EM - 400"."AV409-1".CW.ENABLE := True;
   MachineConfig[8]."Unit Sep"."EM - 400"."AV409-1".ACT_OUT_ADD := 170;
   MachineConfig[8]."Unit Sep"."EM - 400"."FCV409-1".CW.ENABLE := True;
   MachineConfig[8]."Unit Sep"."EM - 400"."FIS409-1".CW.ENABLE := False;
   MachineConfig[8]."Unit Sep"."EM - 400"."FIT409-1".CW.ENABLE := True;
   MachineConfig[8]."Unit Sep"."EM - 400"."TT41X-1".CW.ENABLE := True;
   MachineConfig[8]."Unit Sep"."EM - 400"."TT41X-1"."Type" := 0;
   MachineConfig[8]."Unit Sep"."EM - 400"."TT41X-1".Address := 86;
   MachineConfig[8]."Unit Sep"."EM - 400"."TT41X-1".Min := -50.0;
   MachineConfig[8]."Unit Sep"."EM - 400"."TT41X-1".Max := 150.0;
   MachineConfig[8]."Unit Sep"."EM - 600"."AV63X/441-1".TAG := 'AV441-1';
   MachineConfig[8]."Unit Sep"."EM - 600"."AV63X/441-1".CW.ENABLE := True;
   MachineConfig[8]."Unit Sep"."EM - 600"."AV63X/441-1".CW.NO := False;
   MachineConfig[8]."Unit Sep"."EM - 600"."AV63X/441-1".CW.EXIST := True;
   MachineConfig[8]."Unit Sep"."EM - 600"."AV63X/441-1".ACT_OUT_ADD := 174;
   MachineConfig[8]."Unit Sep"."EM - 701".M701."TYPE" := 2;
   MachineConfig[8]."Unit Sep"."EM - 701".M701.FB_RUN_ADD := 8;
   MachineConfig[8]."Unit Sep"."EM - 701".M701.FB_RDY_ADD := 8;
   MachineConfig[8]."Unit Sep"."EM - 701".M701.OUT_ACT_ADD := 512;
   MachineConfig[8]."Unit Sep"."EM - 701".M701.OUT_RST_ADD := 8;
   MachineConfig[8]."Unit Sep"."EM - 730".TS730.CW.ENABLE := True;
   MachineConfig[8]."Unit Sep"."EM - 730".TS730.Address := 184;
   MachineConfig[8]."Unit Sep"."EM - 740"."P+F PS".Address := 180;
   MachineConfig[8]."Unit Sep"."EM - 740"."P+F OS".Address := 182;
   MachineConfig[8]."Unit Sep"."EM - 740"."P+F ERROR".Address := 183;
   MachineConfig[8]."Unit Sep"."EM - 750".YT75X.Address := 78;
   MachineConfig[8]."Unit Process"."EM - 201"."AV201-1".CW.ENABLE := True;
   MachineConfig[8]."Unit Process"."EM - 201"."AV201-1".CW.FB_CLS_EN := False;
   MachineConfig[8]."Unit Process"."EM - 201"."AV201-1".CW.FB_OPN_EN := False;
   MachineConfig[8]."Unit Process"."EM - 201"."AV201-1".CW.VLV_W_FB := False;
   MachineConfig[8]."Unit Process"."EM - 201"."AV201-1".FB_OPN_ADD := 8;
   MachineConfig[8]."Unit Process"."EM - 201"."AV201-1".FB_CLS_ADD := 8;
   MachineConfig[8]."Unit Process"."EM - 201"."AV201-1".ACT_OUT_ADD := 160;
   MachineConfig[8]."Unit Process"."EM - 201"."FCV201-1".CW.ENABLE := False;
   MachineConfig[8]."Unit Process"."EM - 201"."FIT201-1"."Type" := 0;
   MachineConfig[8]."Unit Process"."EM - 201"."FIT201-1".Address := 88;
   MachineConfig[8]."Unit Process"."EM - 201"."FIT201-1".Max := 50000.0;
   MachineConfig[8]."Unit Process"."EM - 201"."LA201-1".CW.ENABLE := False;
   MachineConfig[8]."Unit Process"."EM - 201"."PIT201-1".CW.ENABLE := True;
   MachineConfig[8]."Unit Process"."EM - 201"."PIT201-1".CW.EXIST := False;
   MachineConfig[8]."Unit Process"."EM - 22X"."AV220-1".CW.ENABLE := True;
   MachineConfig[8]."Unit Process"."EM - 22X"."AV220-1".CW.FB_CLS_EN := False;
   MachineConfig[8]."Unit Process"."EM - 22X"."AV220-1".CW.FB_OPN_EN := False;
   MachineConfig[8]."Unit Process"."EM - 22X"."AV220-1".CW.VLV_W_FB := False;
   MachineConfig[8]."Unit Process"."EM - 22X"."AV220-1".FB_OPN_ADD := 8;
   MachineConfig[8]."Unit Process"."EM - 22X"."AV220-1".FB_CLS_ADD := 8;
   MachineConfig[8]."Unit Process"."EM - 22X"."AV220-1".ACT_OUT_ADD := 162;
   MachineConfig[8]."Unit Process"."EM - 22X"."AV460-1".CW.ENABLE := True;
   MachineConfig[8]."Unit Process"."EM - 22X"."AV460-1".CW.FB_CLS_EN := False;
   MachineConfig[8]."Unit Process"."EM - 22X"."AV460-1".CW.FB_OPN_EN := False;
   MachineConfig[8]."Unit Process"."EM - 22X"."AV460-1".CW.VLV_W_FB := False;
   MachineConfig[8]."Unit Process"."EM - 22X"."AV460-1".FB_OPN_ADD := 8;
   MachineConfig[8]."Unit Process"."EM - 22X"."AV460-1".FB_CLS_ADD := 8;
   MachineConfig[8]."Unit Process"."EM - 22X"."AV460-1".ACT_OUT_ADD := 171;
   MachineConfig[8]."Unit Process"."EM - 22X"."PIT22X-1".CW.ENABLE := True;
   MachineConfig[8]."Unit Process"."EM - 22X"."PIT22X-1".CW.EXIST := False;
   MachineConfig[8]."Unit Process"."EM - 22X"."QT220-1".CW.ENABLE := True;
   MachineConfig[8]."Unit Process"."EM - 22X"."QT220-1".CW.EXIST := False;
   MachineConfig[8]."Unit Process"."EM - 340"."AV340-1".CW.ENABLE := True;
   MachineConfig[8]."Unit Process"."EM - 340"."AV340-1".CW.FB_CLS_EN := False;
   MachineConfig[8]."Unit Process"."EM - 340"."AV340-1".CW.FB_OPN_EN := False;
   MachineConfig[8]."Unit Process"."EM - 340"."AV340-1".CW.VLV_W_FB := False;
   MachineConfig[8]."Unit Process"."EM - 340"."AV340-1".FB_OPN_ADD := 8;
   MachineConfig[8]."Unit Process"."EM - 340"."AV340-1".FB_CLS_ADD := 8;
   MachineConfig[8]."Unit Process"."EM - 340"."AV340-1".ACT_OUT_ADD := 165;
   MachineConfig[8]."Unit Process"."EM - 340"."V340-1".CW.ENABLE := True;
   MachineConfig[8]."Unit Process"."EM - 340"."V340-1".Address := 170;
   MachineConfig[8]."Unit Dch"."EM - 222"."LS222-1".CW.ENABLE := False;
   MachineConfig[8]."Unit Dch"."EM - 222"."P222-1".CW.ENABLE := True;
   MachineConfig[8]."Unit Dch"."EM - 222"."P222-1".CW.EXIST := False;
   MachineConfig[8]."Unit Dch"."EM - 222"."P222-1".FB_RUN_ADD := 194;
   MachineConfig[8]."Unit Dch"."EM - 222"."P222-1".FB_RDY_ADD := 195;
   MachineConfig[8]."Unit Dch"."EM - 222"."P222-1".OUT_ACT_ADD := 182;
   MachineConfig[8]."Unit Dch"."EM - 300"."AV301-1".CW.ENABLE := True;
   MachineConfig[8]."Unit Dch"."EM - 300"."AV301-1".CW.FB_CLS_EN := False;
   MachineConfig[8]."Unit Dch"."EM - 300"."AV301-1".CW.FB_OPN_EN := False;
   MachineConfig[8]."Unit Dch"."EM - 300"."AV301-1".CW.VLV_W_FB := False;
   MachineConfig[8]."Unit Dch"."EM - 300"."AV301-1".FB_OPN_ADD := 8;
   MachineConfig[8]."Unit Dch"."EM - 300"."AV301-1".FB_CLS_ADD := 8;
   MachineConfig[8]."Unit Dch"."EM - 300"."AV301-1".ACT_OUT_ADD := 163;
   MachineConfig[8]."Unit Dch"."EM - 300"."AV320-1".CW.ENABLE := True;
   MachineConfig[8]."Unit Dch"."EM - 300"."AV320-1".CW.FB_CLS_EN := False;
   MachineConfig[8]."Unit Dch"."EM - 300"."AV320-1".CW.FB_OPN_EN := False;
   MachineConfig[8]."Unit Dch"."EM - 300"."AV320-1".CW.VLV_W_FB := False;
   MachineConfig[8]."Unit Dch"."EM - 300"."AV320-1".FB_OPN_ADD := 8;
   MachineConfig[8]."Unit Dch"."EM - 300"."AV320-1".FB_CLS_ADD := 8;
   MachineConfig[8]."Unit Dch"."EM - 300"."AV320-1".ACT_OUT_ADD := 164;
   MachineConfig[8]."Unit Dch"."EM - 375"."AV37X-1".CW.ENABLE := True;
   MachineConfig[8]."Unit Dch"."EM - 375"."AV37X-1".ACT_OUT_ADD := 166;
   MachineConfig[8]."Unit Dch"."EM - 375"."PIS375-1".CW.ENABLE := False;
   MachineConfig[8]."Unit Dch"."EM - 375"."PT37X-1".Tag := 'PT375-1';
   MachineConfig[8]."Unit Dch"."EM - 375"."PT37X-1".CW.ENABLE := True;
   MachineConfig[8]."Unit Dch"."EM - 375"."PT37X-1".Address := 76;
   MachineConfig[8]."Unit Dch"."EM - 375"."PT37X-1".Max := 600.0;
   MachineConfig[8]."Unit Dch"."EM - 506".IP506a.CW.ENABLE := True;
   MachineConfig[8]."Unit Dch"."EM - 506".AVDCH.TAG := '506b';
   MachineConfig[8]."Unit Dch"."EM - 506".AVDCH.ACT_OUT_ADD := 167;
   MachineConfig[8].Options."EM - P201"."P201-1".FB_RUN_ADD := 196;
   MachineConfig[8].Options."EM - P201"."P201-1".FB_RDY_ADD := 197;
   MachineConfig[8].Options."EM - P201"."P201-1".OUT_ACT_ADD := 183;
   MachineConfig[8].Options."EM - P201"."P201-1".OUT_RST_ADD := 184;
   MachineConfig[8].Options."EM - P201"."P201-1_SPEED_REF".Address := 70;
   MachineConfig[9].Machine."Family" := 2;
   MachineConfig[9].Machine.TypeNo := 29;
   MachineConfig[9].Machine.Range := 2;
   MachineConfig[9].Machine.SepType := 1;
   MachineConfig[9].Machine.Frame := 1;
   MachineConfig[9].Machine.DchSystem := 2;
   MachineConfig[9].Machine.Spare_1 := 3;
   MachineConfig[9].Machine.FeedPump := 1;
   MachineConfig[9].Machine.Spare_2 := 2;
   MachineConfig[9].Machine.ConditionAlert := 1;
   MachineConfig[9].Machine.eWON := 1;
   MachineConfig[9]."Unit Sep"."EM - 100"."L-YELLOW".CW.ENABLE := false;
   MachineConfig[9]."Unit Sep"."EM - 400"."AV409-1".CW.ENABLE := TRUE;
   MachineConfig[9]."Unit Sep"."EM - 400"."FCV409-1".CW.ENABLE := True;
   MachineConfig[9]."Unit Sep"."EM - 400"."FIT409-1".CW.ENABLE := True;
   MachineConfig[9]."Unit Sep"."EM - 400"."TT41X-1".CW.ENABLE := True;
   MachineConfig[9]."Unit Sep"."EM - 400"."TT41X-1".Address := 142;
   MachineConfig[9]."Unit Sep"."EM - 600"."AV63X/441-1".TAG := 'AV441-1';
   MachineConfig[9]."Unit Sep"."EM - 600"."AV63X/441-1".CW.ENABLE := True;
   MachineConfig[9]."Unit Sep"."EM - 600"."AV63X/441-1".CW.NO := False;
   MachineConfig[9]."Unit Sep"."EM - 600"."AV63X/441-1".CW.EXIST := True;
   MachineConfig[9]."Unit Sep"."EM - 600"."AV63X/441-1".ACT_OUT_ADD := 331;
   MachineConfig[9]."Unit Sep"."EM - 600"."FIS615-1".CW.ENABLE := False;
   MachineConfig[9]."Unit Sep"."EM - 730".TS730.CW.ENABLE := true;
   MachineConfig[9]."Unit Sep"."EM - 730".TT731a.CW.ENABLE := True;
   MachineConfig[9]."Unit Sep"."EM - 730".TT733.CW.ENABLE := True;
   MachineConfig[9]."Unit Sep"."EM - 750".YT75X.CW.ENABLE := TRUE;
   MachineConfig[9]."Unit Process"."EM - 201"."AV201-1".CW.ENABLE := True;
   MachineConfig[9]."Unit Process"."EM - 201"."FIT201-1"."Type" := 2;
   MachineConfig[9]."Unit Process"."EM - 201"."FIT201-1".Address := 256;
   MachineConfig[9]."Unit Process"."EM - 201"."FIT201-1".Max := 65000.0;
   MachineConfig[9]."Unit Process"."EM - 201"."QT201-1".CW.ENABLE := True;
   MachineConfig[9]."Unit Process"."EM - 22X"."AV220-1".CW.ENABLE := True;
   MachineConfig[9]."Unit Process"."EM - 22X"."AV460-1".CW.ENABLE := True;
   MachineConfig[9]."Unit Process"."EM - 22X"."FIT22X-1".CW.ENABLE := True;
   MachineConfig[9]."Unit Process"."EM - 22X"."FIT22X-1".CW.EXIST := false;
   MachineConfig[9]."Unit Process"."EM - 22X"."QT220-1".Tag := 'QT220-1';
   MachineConfig[9]."Unit Process"."EM - 22X"."QT220-1".CW.ENABLE := True;
   MachineConfig[9]."Unit Process"."EM - 22X"."QT220-1".CW.EXIST := False;
   MachineConfig[9]."Unit Process"."EM - 22X"."QT220-1".Address := 70;
   MachineConfig[9]."Unit Process"."EM - 22X"."LA220-1".CW.ENABLE := True;
   MachineConfig[9]."Unit Process"."EM - 340"."AV340-1".CW.ENABLE := True;
   MachineConfig[9]."Unit Process"."EM - 340"."AV340-2".CW.ENABLE := True;
   MachineConfig[9]."Unit Process"."EM - 340"."AV460-2".CW.ENABLE := True;
   MachineConfig[9]."Unit Process"."EM - 340"."PIS340-1".CW.ENABLE := True;
   MachineConfig[9]."Unit Dch"."EM - 222"."LS222-1".CW.EXIST := False;
   MachineConfig[9]."Unit Dch"."EM - 222"."P222-1".CW.EXIST := False;
   MachineConfig[9]."Unit Dch"."EM - 222"."TS222-1".CW.ENABLE := true;
   MachineConfig[9]."Unit Dch"."EM - 300"."AV301-1".CW.ENABLE := True;
   MachineConfig[9]."Unit Dch"."EM - 300"."AV302-1".CW.ENABLE := True;
   MachineConfig[9]."Unit Dch"."EM - 300"."AV303-1".CW.ENABLE := True;
   MachineConfig[9]."Unit Dch"."EM - 300"."AV304-1".CW.ENABLE := True;
   MachineConfig[9]."Unit Dch"."EM - 300"."AV305-1".CW.ENABLE := True;
   MachineConfig[9]."Unit Dch"."EM - 300"."AV306-1".CW.ENABLE := True;
   MachineConfig[9]."Unit Dch"."EM - 300"."AV320-1".CW.ENABLE := True;
   MachineConfig[9]."Unit Dch"."EM - 375"."AV37X-1".CW.ENABLE := True;
   MachineConfig[9]."Unit Dch"."EM - 506".IP506a.CW.ENABLE := True;
   MachineConfig[9]."Unit Dch"."EM - 506".AVDCH.CW.ENABLE := true;
   MachineConfig[10].Machine."Family" := 2;
   MachineConfig[10].Machine.TypeNo := 30;
   MachineConfig[10].Machine.Range := 2;
   MachineConfig[10].Machine.SepType := 1;
   MachineConfig[10].Machine.Frame := 1;
   MachineConfig[10].Machine.DchSystem := 2;
   MachineConfig[10].Machine.Spare_1 := 3;
   MachineConfig[10].Machine.FeedPump := 1;
   MachineConfig[10].Machine.Spare_2 := 2;
   MachineConfig[10].Machine.ConditionAlert := 1;
   MachineConfig[10].Machine.eWON := 1;
   MachineConfig[10]."Unit Sep"."EM - 100"."L-YELLOW".CW.ENABLE := false;
   MachineConfig[10]."Unit Sep"."EM - 400"."AV409-1".CW.ENABLE := True;
   MachineConfig[10]."Unit Sep"."EM - 400"."FCV409-1".CW.ENABLE := True;
   MachineConfig[10]."Unit Sep"."EM - 400"."FIT409-1".CW.ENABLE := True;
   MachineConfig[10]."Unit Sep"."EM - 400"."TT41X-1".CW.ENABLE := True;
   MachineConfig[10]."Unit Sep"."EM - 400"."TT41X-1".Address := 142;
   MachineConfig[10]."Unit Sep"."EM - 600"."AV615-1".CW.ENABLE := True;
   MachineConfig[10]."Unit Sep"."EM - 600"."FIS615-1".Tag := 'FIS635a-1';
   MachineConfig[10]."Unit Sep"."EM - 600"."FIS615-1".CW.ENABLE := True;
   MachineConfig[10]."Unit Sep"."EM - 600"."FIS635-1".Tag := 'FIS635b-1';
   MachineConfig[10]."Unit Sep"."EM - 600"."FIS635-1".CW.ENABLE := True;
   MachineConfig[10]."Unit Sep"."EM - 730".TS730.CW.ENABLE := true;
   MachineConfig[10]."Unit Sep"."EM - 730".TT731a.CW.ENABLE := True;
   MachineConfig[10]."Unit Sep"."EM - 730".TT733.CW.ENABLE := True;
   MachineConfig[10]."Unit Sep"."EM - 750".YT75X.CW.ENABLE := TRUE;
   MachineConfig[10]."Unit Process"."EM - 201"."AV201-1".CW.ENABLE := True;
   MachineConfig[10]."Unit Process"."EM - 201"."FIT201-1"."Type" := 2;
   MachineConfig[10]."Unit Process"."EM - 201"."FIT201-1".Address := 256;
   MachineConfig[10]."Unit Process"."EM - 201"."FIT201-1".Max := 65000.0;
   MachineConfig[10]."Unit Process"."EM - 201"."QT201-1".CW.ENABLE := True;
   MachineConfig[10]."Unit Process"."EM - 22X"."AV220-1".CW.ENABLE := True;
   MachineConfig[10]."Unit Process"."EM - 22X"."AV460-1".CW.ENABLE := True;
   MachineConfig[10]."Unit Process"."EM - 22X"."FIT22X-1".CW.ENABLE := True;
   MachineConfig[10]."Unit Process"."EM - 22X"."FIT22X-1".CW.EXIST := false;
   MachineConfig[10]."Unit Process"."EM - 22X"."FIT22X-1".Address := 276;
   MachineConfig[10]."Unit Process"."EM - 22X"."QT220-1".CW.ENABLE := True;
   MachineConfig[10]."Unit Process"."EM - 22X"."QT220-1".CW.EXIST := false;
   MachineConfig[10]."Unit Process"."EM - 22X"."LA220-1".CW.ENABLE := True;
   MachineConfig[10]."Unit Process"."EM - 340"."AV340-1".CW.ENABLE := True;
   MachineConfig[10]."Unit Process"."EM - 340"."AV340-2".CW.ENABLE := True;
   MachineConfig[10]."Unit Process"."EM - 340"."AV460-2".CW.ENABLE := True;
   MachineConfig[10]."Unit Process"."EM - 340"."PIS340-1".CW.ENABLE := True;
   MachineConfig[10]."Unit Dch"."EM - 222"."LS222-1".CW.EXIST := False;
   MachineConfig[10]."Unit Dch"."EM - 222"."P222-1".CW.EXIST := False;
   MachineConfig[10]."Unit Dch"."EM - 222"."TS222-1".CW.ENABLE := true;
   MachineConfig[10]."Unit Dch"."EM - 300"."AV301-1".CW.ENABLE := True;
   MachineConfig[10]."Unit Dch"."EM - 300"."AV303-1".CW.ENABLE := True;
   MachineConfig[10]."Unit Dch"."EM - 300"."AV304-1".CW.ENABLE := True;
   MachineConfig[10]."Unit Dch"."EM - 300"."AV305-1".CW.ENABLE := True;
   MachineConfig[10]."Unit Dch"."EM - 300"."AV320-1".CW.ENABLE := True;
   MachineConfig[10]."Unit Dch"."EM - 300"."AV635-1".CW.ENABLE := True;
   MachineConfig[10]."Unit Dch"."EM - 375"."AV37X-1".CW.ENABLE := True;
   MachineConfig[10]."Unit Dch"."EM - 506".IP506a.CW.ENABLE := True;
   MachineConfig[10]."Unit Dch"."EM - 506".AVDCH.CW.ENABLE := true;
   MachineConfig[11].Machine."Family" := 2;
   MachineConfig[11].Machine.TypeNo := 31;
   MachineConfig[11].Machine.Range := 1;
   MachineConfig[11].Machine.SepType := 1;
   MachineConfig[11].Machine.Frame := 1;
   MachineConfig[11].Machine.DchSystem := 2;
   MachineConfig[11].Machine.Spare_1 := 2;
   MachineConfig[11].Machine.FeedPump := 1;
   MachineConfig[11].Machine.Spare_2 := 2;
   MachineConfig[11].Machine.eMotion := 1;
   MachineConfig[11].Machine.ConditionAlert := 1;
   MachineConfig[11].Machine.eWON := 1;
   MachineConfig[11]."Unit Sep"."EM - 100"."L-YELLOW".CW.ENABLE := false;
   MachineConfig[11]."Unit Sep"."EM - 400"."AV409-1".CW.ENABLE := True;
   MachineConfig[11]."Unit Sep"."EM - 400"."FCV409-1".CW.ENABLE := True;
   MachineConfig[11]."Unit Sep"."EM - 400"."FIT409-1".CW.ENABLE := True;
   MachineConfig[11]."Unit Sep"."EM - 400"."TT41X-1".Tag := 'TT410-1';
   MachineConfig[11]."Unit Sep"."EM - 400"."TT41X-1".CW.ENABLE := True;
   MachineConfig[11]."Unit Sep"."EM - 400"."TT41X-1".Address := 142;
   MachineConfig[11]."Unit Sep"."EM - 600"."AV615-1".CW.ENABLE := True;
   MachineConfig[11]."Unit Sep"."EM - 600"."FIS615-1".CW.ENABLE := True;
   MachineConfig[11]."Unit Sep"."EM - 600"."FIS635-1".CW.ENABLE := True;
   MachineConfig[11]."Unit Sep"."EM - 730".TS730.CW.ENABLE := true;
   MachineConfig[11]."Unit Sep"."EM - 730".TT731a.CW.ENABLE := True;
   MachineConfig[11]."Unit Sep"."EM - 730".TT733.CW.ENABLE := True;
   MachineConfig[11]."Unit Sep"."EM - 750".YT75X.CW.ENABLE := TRUE;
   MachineConfig[11]."Unit Process"."EM - 201"."AV201-1".CW.ENABLE := True;
   MachineConfig[11]."Unit Process"."EM - 201"."FIT201-1"."Type" := 2;
   MachineConfig[11]."Unit Process"."EM - 201"."FIT201-1".Address := 256;
   MachineConfig[11]."Unit Process"."EM - 201"."FIT201-1".Max := 65000.0;
   MachineConfig[11]."Unit Process"."EM - 201"."QT201-1".CW.ENABLE := True;
   MachineConfig[11]."Unit Process"."EM - 22X"."AV220-1".CW.ENABLE := True;
   MachineConfig[11]."Unit Process"."EM - 22X"."AV460-1".CW.ENABLE := True;
   MachineConfig[11]."Unit Process"."EM - 22X"."FIT22X-1".CW.ENABLE := True;
   MachineConfig[11]."Unit Process"."EM - 22X"."FIT22X-1".CW.EXIST := false;
   MachineConfig[11]."Unit Process"."EM - 22X"."FIT22X-1".Address := 276;
   MachineConfig[11]."Unit Process"."EM - 22X"."QT220-1".CW.ENABLE := True;
   MachineConfig[11]."Unit Process"."EM - 22X"."QT220-1".CW.EXIST := false;
   MachineConfig[11]."Unit Process"."EM - 22X"."LA220-1".CW.ENABLE := True;
   MachineConfig[11]."Unit Process"."EM - 340"."AV340-1".CW.ENABLE := True;
   MachineConfig[11]."Unit Process"."EM - 340"."AV340-2".CW.ENABLE := True;
   MachineConfig[11]."Unit Process"."EM - 340"."AV460-2".CW.ENABLE := True;
   MachineConfig[11]."Unit Process"."EM - 340"."PIS340-1".CW.ENABLE := True;
   MachineConfig[11]."Unit Dch"."EM - 222"."P222-1".CW.EXIST := False;
   MachineConfig[11]."Unit Dch"."EM - 222"."TS222-1".CW.ENABLE := true;
   MachineConfig[11]."Unit Dch"."EM - 300"."AV301-1".CW.ENABLE := True;
   MachineConfig[11]."Unit Dch"."EM - 300"."AV303-1".CW.ENABLE := True;
   MachineConfig[11]."Unit Dch"."EM - 300"."AV304-1".CW.ENABLE := True;
   MachineConfig[11]."Unit Dch"."EM - 300"."AV305-1".CW.ENABLE := True;
   MachineConfig[11]."Unit Dch"."EM - 300"."AV320-1".CW.ENABLE := True;
   MachineConfig[11]."Unit Dch"."EM - 300"."AV635-1".CW.ENABLE := True;
   MachineConfig[11]."Unit Dch"."EM - 375"."AV37X-1".CW.ENABLE := True;
   MachineConfig[11]."Unit Dch"."EM - 375"."PT37X-1".CW.ENABLE := True;
   MachineConfig[11]."Unit Dch"."EM - 375"."PT37X-1".CW.EXIST := False;
   MachineConfig[11]."Unit Dch"."EM - 506"."AV543-1".CW.ENABLE := True;
   MachineConfig[11]."Unit Dch"."EM - 506"."AV543-1".CW.EXIST := False;
   MachineConfig[11]."Unit Dch"."EM - 506".IP506a.CW.ENABLE := True;
   MachineConfig[11]."Unit Dch"."EM - 506"."PV376-1".CW.ENABLE := True;
   MachineConfig[11]."Unit Dch"."EM - 506"."PV376-1".CW.EXIST := False;
   MachineConfig[11]."Unit Dch"."EM - 506"."PV376-2".CW.ENABLE := True;
   MachineConfig[11]."Unit Dch"."EM - 506"."PV376-2".CW.EXIST := False;
   MachineConfig[11]."Unit Dch"."EM - 506".AVDCH.CW.ENABLE := true;
   MachineConfig[12].Machine."Family" := 2;
   MachineConfig[12].Machine.TypeNo := 32;
   MachineConfig[12].Machine.Range := 1;
   MachineConfig[12].Machine.SepType := 1;
   MachineConfig[12].Machine.Frame := 1;
   MachineConfig[12].Machine.DchSystem := 2;
   MachineConfig[12].Machine.Spare_1 := 2;
   MachineConfig[12].Machine.FeedPump := 1;
   MachineConfig[12].Machine.Spare_2 := 2;
   MachineConfig[12].Machine.eMotion := 1;
   MachineConfig[12].Machine.ConditionAlert := 1;
   MachineConfig[12].Machine.eWON := 1;
   MachineConfig[12]."Unit Sep"."EM - 100"."L-YELLOW".CW.ENABLE := false;
   MachineConfig[12]."Unit Sep"."EM - 100"."CA VIB WARN".CW.ENABLE := True;
   MachineConfig[12]."Unit Sep"."EM - 100"."CA VIB ALM".CW.ENABLE := True;
   MachineConfig[12]."Unit Sep"."EM - 100"."CA ERROR".CW.ENABLE := True;
   MachineConfig[12]."Unit Sep"."EM - 100"."CA WD".CW.ENABLE := True;
   MachineConfig[12]."Unit Sep"."EM - 400"."AV409-1".CW.ENABLE := True;
   MachineConfig[12]."Unit Sep"."EM - 400"."FCV409-1".CW.ENABLE := True;
   MachineConfig[12]."Unit Sep"."EM - 400"."FIT409-1".CW.ENABLE := True;
   MachineConfig[12]."Unit Sep"."EM - 400"."TT41X-1".CW.ENABLE := True;
   MachineConfig[12]."Unit Sep"."EM - 400"."TT41X-1".Address := 142;
   MachineConfig[12]."Unit Sep"."EM - 600"."AV615-1".CW.ENABLE := True;
   MachineConfig[12]."Unit Sep"."EM - 600"."FIS615-1".CW.ENABLE := True;
   MachineConfig[12]."Unit Sep"."EM - 600"."FIS635-1".CW.ENABLE := True;
   MachineConfig[12]."Unit Sep"."EM - 730".TS730.CW.ENABLE := true;
   MachineConfig[12]."Unit Sep"."EM - 730".TT731a.CW.ENABLE := True;
   MachineConfig[12]."Unit Sep"."EM - 730".TT733.CW.ENABLE := True;
   MachineConfig[12]."Unit Sep"."EM - 750".YT75X.CW.ENABLE := TRUE;
   MachineConfig[12]."Unit Process"."EM - 201"."AV201-1".CW.ENABLE := True;
   MachineConfig[12]."Unit Process"."EM - 201"."FIT201-1"."Type" := 2;
   MachineConfig[12]."Unit Process"."EM - 201"."FIT201-1".Address := 256;
   MachineConfig[12]."Unit Process"."EM - 201"."FIT201-1".Max := 65000.0;
   MachineConfig[12]."Unit Process"."EM - 201"."QT201-1".CW.ENABLE := True;
   MachineConfig[12]."Unit Process"."EM - 22X"."AV220-1".CW.ENABLE := True;
   MachineConfig[12]."Unit Process"."EM - 22X"."AV460-1".CW.ENABLE := True;
   MachineConfig[12]."Unit Process"."EM - 22X"."FIT22X-1".CW.ENABLE := True;
   MachineConfig[12]."Unit Process"."EM - 22X"."FIT22X-1".Address := 276;
   MachineConfig[12]."Unit Process"."EM - 22X"."QT220-1".Tag := 'QT220-1';
   MachineConfig[12]."Unit Process"."EM - 22X"."QT220-1".CW.ENABLE := True;
   MachineConfig[12]."Unit Process"."EM - 22X"."QT220-1".CW.EXIST := false;
   MachineConfig[12]."Unit Process"."EM - 22X"."LA220-1".CW.ENABLE := True;
   MachineConfig[12]."Unit Process"."EM - 340"."AV340-1".CW.ENABLE := True;
   MachineConfig[12]."Unit Process"."EM - 340"."AV340-2".CW.ENABLE := True;
   MachineConfig[12]."Unit Process"."EM - 340"."AV460-2".CW.ENABLE := True;
   MachineConfig[12]."Unit Dch"."EM - 222"."P222-1".CW.EXIST := False;
   MachineConfig[12]."Unit Dch"."EM - 222"."TS222-1".CW.ENABLE := true;
   MachineConfig[12]."Unit Dch"."EM - 300"."AV301-1".CW.ENABLE := True;
   MachineConfig[12]."Unit Dch"."EM - 300"."AV302-1".CW.ENABLE := True;
   MachineConfig[12]."Unit Dch"."EM - 300"."AV303-1".CW.ENABLE := True;
   MachineConfig[12]."Unit Dch"."EM - 300"."AV304-1".CW.ENABLE := True;
   MachineConfig[12]."Unit Dch"."EM - 300"."AV305-1".CW.ENABLE := True;
   MachineConfig[12]."Unit Dch"."EM - 300"."AV320-1".CW.ENABLE := True;
   MachineConfig[12]."Unit Dch"."EM - 300"."AV635-1".CW.ENABLE := True;
   MachineConfig[12]."Unit Dch"."EM - 375"."AV37X-1".CW.ENABLE := True;
   MachineConfig[12]."Unit Dch"."EM - 375"."PT37X-1".CW.ENABLE := True;
   MachineConfig[12]."Unit Dch"."EM - 375"."PT37X-1".CW.EXIST := False;
   MachineConfig[12]."Unit Dch"."EM - 506"."AV543-1".CW.ENABLE := True;
   MachineConfig[12]."Unit Dch"."EM - 506"."AV543-1".CW.EXIST := False;
   MachineConfig[12]."Unit Dch"."EM - 506".IP506a.CW.ENABLE := True;
   MachineConfig[12]."Unit Dch"."EM - 506"."PV376-1".CW.ENABLE := True;
   MachineConfig[12]."Unit Dch"."EM - 506"."PV376-1".CW.EXIST := False;
   MachineConfig[12]."Unit Dch"."EM - 506"."PV376-2".CW.ENABLE := True;
   MachineConfig[12]."Unit Dch"."EM - 506"."PV376-2".CW.EXIST := False;
   MachineConfig[12]."Unit Dch"."EM - 506".AVDCH.CW.ENABLE := true;
   MachineConfig[13].Machine."Family" := 2;
   MachineConfig[13].Machine.TypeNo := 33;
   MachineConfig[13].Machine.Range := 1;
   MachineConfig[13].Machine.SepType := 1;
   MachineConfig[13].Machine.Frame := 1;
   MachineConfig[13].Machine.DchSystem := 2;
   MachineConfig[13].Machine.Spare_1 := 2;
   MachineConfig[13].Machine.FeedPump := 1;
   MachineConfig[13].Machine.Spare_2 := 2;
   MachineConfig[13].Machine.ConditionAlert := 1;
   MachineConfig[13].Machine.eWON := 1;
   MachineConfig[13]."Unit Sep"."EM - 100"."L-YELLOW".CW.ENABLE := false;
   MachineConfig[13]."Unit Sep"."EM - 400"."AV409-1".CW.ENABLE := True;
   MachineConfig[13]."Unit Sep"."EM - 400"."FCV409-1".CW.ENABLE := True;
   MachineConfig[13]."Unit Sep"."EM - 400"."FIT409-1".CW.ENABLE := True;
   MachineConfig[13]."Unit Sep"."EM - 400"."TT41X-1".CW.ENABLE := True;
   MachineConfig[13]."Unit Sep"."EM - 400"."TT41X-1".Address := 142;
   MachineConfig[13]."Unit Sep"."EM - 600"."AV615-1".CW.ENABLE := True;
   MachineConfig[13]."Unit Sep"."EM - 600"."AV63X/441-1".TAG := 'AV441-1';
   MachineConfig[13]."Unit Sep"."EM - 600"."AV63X/441-1".CW.ENABLE := True;
   MachineConfig[13]."Unit Sep"."EM - 600"."AV63X/441-1".ACT_OUT_ADD := 331;
   MachineConfig[13]."Unit Sep"."EM - 600"."FIS615-1".CW.ENABLE := True;
   MachineConfig[13]."Unit Sep"."EM - 730".TS730.CW.ENABLE := true;
   MachineConfig[13]."Unit Sep"."EM - 730".TT731a.CW.ENABLE := True;
   MachineConfig[13]."Unit Sep"."EM - 730".TT733.CW.ENABLE := True;
   MachineConfig[13]."Unit Sep"."EM - 750".YT75X.CW.ENABLE := TRUE;
   MachineConfig[13]."Unit Process"."EM - 201"."AV201-1".CW.ENABLE := True;
   MachineConfig[13]."Unit Process"."EM - 201"."FIT201-1"."Type" := 2;
   MachineConfig[13]."Unit Process"."EM - 201"."FIT201-1".Address := 256;
   MachineConfig[13]."Unit Process"."EM - 201"."FIT201-1".Max := 65000.0;
   MachineConfig[13]."Unit Process"."EM - 201"."QT201-1".CW.ENABLE := True;
   MachineConfig[13]."Unit Process"."EM - 22X"."AV220-1".CW.ENABLE := True;
   MachineConfig[13]."Unit Process"."EM - 22X"."AV460-1".CW.ENABLE := True;
   MachineConfig[13]."Unit Process"."EM - 22X"."FIT22X-1".CW.ENABLE := True;
   MachineConfig[13]."Unit Process"."EM - 22X"."FIT22X-1".CW.EXIST := false;
   MachineConfig[13]."Unit Process"."EM - 22X"."FIT22X-1".Address := 276;
   MachineConfig[13]."Unit Process"."EM - 22X"."QT220-1".Tag := 'QT220-1';
   MachineConfig[13]."Unit Process"."EM - 22X"."QT220-1".CW.ENABLE := True;
   MachineConfig[13]."Unit Process"."EM - 22X"."QT220-1".CW.EXIST := False;
   MachineConfig[13]."Unit Process"."EM - 22X"."LA220-1".CW.ENABLE := True;
   MachineConfig[13]."Unit Process"."EM - 340"."AV340-1".CW.ENABLE := True;
   MachineConfig[13]."Unit Process"."EM - 340"."AV340-2".CW.ENABLE := True;
   MachineConfig[13]."Unit Process"."EM - 340"."AV460-2".CW.ENABLE := True;
   MachineConfig[13]."Unit Dch"."EM - 222"."LS222-1".CW.ENABLE := True;
   MachineConfig[13]."Unit Dch"."EM - 222"."LS222-1".CW.EXIST := False;
   MachineConfig[13]."Unit Dch"."EM - 222"."P222-1".CW.EXIST := False;
   MachineConfig[13]."Unit Dch"."EM - 222"."TS222-1".CW.ENABLE := true;
   MachineConfig[13]."Unit Dch"."EM - 300"."AV301-1".CW.ENABLE := True;
   MachineConfig[13]."Unit Dch"."EM - 300"."AV303-1".CW.ENABLE := True;
   MachineConfig[13]."Unit Dch"."EM - 300"."AV304-1".CW.ENABLE := True;
   MachineConfig[13]."Unit Dch"."EM - 300"."AV305-1".CW.ENABLE := True;
   MachineConfig[13]."Unit Dch"."EM - 300"."AV320-1".CW.ENABLE := True;
   MachineConfig[13]."Unit Dch"."EM - 300"."AV635-1".TAG := 'AV441-1';
   MachineConfig[13]."Unit Dch"."EM - 300"."AV635-1".CW.ENABLE := True;
   MachineConfig[13]."Unit Dch"."EM - 375"."AV37X-1".CW.ENABLE := True;
   MachineConfig[13]."Unit Dch"."EM - 506".IP506a.CW.ENABLE := True;
   MachineConfig[13]."Unit Dch"."EM - 506".AVDCH.CW.ENABLE := true;
   MachineConfig[14].Machine."Family" := 2;
   MachineConfig[14].Machine.TypeNo := 34;
   MachineConfig[14].Machine.Range := 1;
   MachineConfig[14].Machine.SepType := 1;
   MachineConfig[14].Machine.Frame := 1;
   MachineConfig[14].Machine.DchSystem := 2;
   MachineConfig[14].Machine.Spare_1 := 2;
   MachineConfig[14].Machine.FeedPump := 1;
   MachineConfig[14].Machine.Spare_2 := 2;
   MachineConfig[14].Machine.eMotion := 1;
   MachineConfig[14].Machine.ConditionAlert := 1;
   MachineConfig[14].Machine.eWON := 1;
   MachineConfig[14]."Unit Sep"."EM - 100"."L-YELLOW".CW.ENABLE := false;
   MachineConfig[14]."Unit Sep"."EM - 100"."CA VIB WARN".CW.ENABLE := True;
   MachineConfig[14]."Unit Sep"."EM - 100"."CA VIB ALM".CW.ENABLE := True;
   MachineConfig[14]."Unit Sep"."EM - 100"."CA ERROR".CW.ENABLE := True;
   MachineConfig[14]."Unit Sep"."EM - 100"."CA WD".CW.ENABLE := True;
   MachineConfig[14]."Unit Sep"."EM - 400"."AV409-1".CW.ENABLE := True;
   MachineConfig[14]."Unit Sep"."EM - 400"."FCV409-1".CW.ENABLE := True;
   MachineConfig[14]."Unit Sep"."EM - 400"."FIT409-1".CW.ENABLE := True;
   MachineConfig[14]."Unit Sep"."EM - 400"."TT41X-1".Tag := 'TT410-1';
   MachineConfig[14]."Unit Sep"."EM - 400"."TT41X-1".CW.ENABLE := True;
   MachineConfig[14]."Unit Sep"."EM - 600"."AV615-1".CW.ENABLE := True;
   MachineConfig[14]."Unit Sep"."EM - 600"."AV63X/441-1".TAG := 'AV635-1';
   MachineConfig[14]."Unit Sep"."EM - 600"."AV63X/441-1".CW.ENABLE := True;
   MachineConfig[14]."Unit Sep"."EM - 600"."AV63X/441-1".CW.EXIST := True;
   MachineConfig[14]."Unit Sep"."EM - 600"."FIS615-1".CW.ENABLE := True;
   MachineConfig[14]."Unit Sep"."EM - 600"."FIS635-1".CW.ENABLE := True;
   MachineConfig[14]."Unit Sep"."EM - 730".TS730.CW.ENABLE := true;
   MachineConfig[14]."Unit Sep"."EM - 730".TT731a.CW.ENABLE := True;
   MachineConfig[14]."Unit Sep"."EM - 730".TT733.CW.ENABLE := True;
   MachineConfig[14]."Unit Sep"."EM - 750".YT75X.CW.ENABLE := TRUE;
   MachineConfig[14]."Unit Process"."EM - 201"."AV201-1".CW.ENABLE := True;
   MachineConfig[14]."Unit Process"."EM - 201"."FIT201-1"."Type" := 2;
   MachineConfig[14]."Unit Process"."EM - 201"."FIT201-1".Address := 256;
   MachineConfig[14]."Unit Process"."EM - 201"."FIT201-1".Max := 65000.0;
   MachineConfig[14]."Unit Process"."EM - 201"."QT201-1".CW.ENABLE := True;
   MachineConfig[14]."Unit Process"."EM - 22X"."AV220-1".CW.ENABLE := True;
   MachineConfig[14]."Unit Process"."EM - 22X"."AV460-1".CW.ENABLE := True;
   MachineConfig[14]."Unit Process"."EM - 22X"."FIT22X-1".CW.ENABLE := True;
   MachineConfig[14]."Unit Process"."EM - 22X"."FIT22X-1".CW.EXIST := false;
   MachineConfig[14]."Unit Process"."EM - 22X"."FIT22X-1".Address := 276;
   MachineConfig[14]."Unit Process"."EM - 22X"."QT220-1".Tag := 'QT220-1';
   MachineConfig[14]."Unit Process"."EM - 22X"."QT220-1".CW.ENABLE := True;
   MachineConfig[14]."Unit Process"."EM - 22X"."QT220-1".CW.EXIST := false;
   MachineConfig[14]."Unit Process"."EM - 22X"."QT220-1".Address := 70;
   MachineConfig[14]."Unit Process"."EM - 22X"."LA220-1".CW.ENABLE := True;
   MachineConfig[14]."Unit Process"."EM - 340"."AV340-1".CW.ENABLE := True;
   MachineConfig[14]."Unit Process"."EM - 340"."AV340-2".CW.ENABLE := True;
